// TIA Portal V20 export
DATA_BLOCK "HmiInterface"   // DB93
{ DB_Accessible_From_OPC_UA := 'FALSE' }
AUTHOR : ERsystem_FA2_DH. Kim
// stored: Access Published, DBAccessibleFromOPCUA false, DBAccessibleFromWebserver false, MemoryReserve 100, Namespace Unit1.Em6
   VAR
      em : "LAF_typeEmInterface";
      cm : Struct
         softCam : "Unit1.type_emRelations_em6_SoftCam";
         brakeTest : Struct
            mendrelAnodeFrontAxisZ : "LER_typeBrakeTestEmInterface";
            mendrelAnodeRearAxisZ : "LER_typeBrakeTestEmInterface";
            mendrelCathodeFrontAxisZ : "LER_typeBrakeTestEmInterface";
            mendrelCathodeRearAxisZ : "LER_typeBrakeTestEmInterface";
            stackTableAxisZ : "LER_typeBrakeTestEmInterface";
            stackTableOutFrontAxisZ : "LER_typeBrakeTestEmInterface";
            stackTableOutRearAxisZ : "LER_typeBrakeTestEmInterface";
         END_STRUCT;
         gearIn : Struct
            finalRollerAxisX : "LER_typeGearInInterface";
            stackTableOutAxisZ : "LER_typeGearInInterface";
         END_STRUCT;
      END_STRUCT;
      motion : Struct
         jobs { S7_SetPoint := 'True'} : "LAF_typeJobsInterface";
         sequence { S7_SetPoint := 'True'} : "LAF_typeSequenceInterface";
      END_STRUCT;
      stackTable : Struct
         jobs { S7_SetPoint := 'True'} : "LAF_typeJobsInterface";
         sequence { S7_SetPoint := 'True'} : "LAF_typeSequenceInterface";
      END_STRUCT;
      gaugeRnR : Struct
         jobs { S7_SetPoint := 'True'} : "LAF_typeJobsInterface";
         sequence { S7_SetPoint := 'True'} : "LAF_typeSequenceInterface";
      END_STRUCT;
      utility : Struct
         jobs { S7_SetPoint := 'True'} : "LAF_typeJobsInterface";
         sequence { S7_SetPoint := 'True'} : "LAF_typeSequenceInterface";
      END_STRUCT;
      recipe : Struct
         anodeThickness : LReal := 0.0;
         cathodeThickness : LReal := 0.0;
         sepaThickenss : LReal := 0.0;
         jellyRollThickness : LReal := 0.0;
      END_STRUCT;
      auxiliary : Struct
         parameters : Struct
            finalRollerFrontHomeOffset : LReal := 0.0;
            finalRollerRearHomeOffset : LReal := 0.0;
            stackTableOutFrontHomeOffset : LReal := 0.0;
            stackTableOutRearHomeOffset : LReal := 0.0;
         END_STRUCT;
         commands : Struct
            finalRollerHome : Bool := FALSE;
            stackTableOutHome : Bool := FALSE;
            allMendrelOpen : Bool := FALSE;
            allMendrelClose : Bool := FALSE;
         END_STRUCT;
         monitoring : Struct
            Null : Bool := FALSE;
         END_STRUCT;
      END_STRUCT;
      cmStackTableElectrodeDetect { S7_SetPoint := 'True'} : "LBC_typeDigitalSignalInterface";
   END_VAR
   VAR RETAIN
      cmMasterVirtualAxisX { ExternalVisible := 'False'; ExternalWritable := 'False'} : "LBC_typeAxis64PosInterface";
      cmFinalRollerFrontAxisX { S7_SetPoint := 'True'} : "LBC_typeAxis64PosInterface";
      cmFinalRollerRearAxisX { S7_SetPoint := 'True'} : "LBC_typeAxis64PosInterface";
      cmMendrelAnodeFrontAxisY { S7_SetPoint := 'True'} : "LBC_typeAxis64PosInterface";
      cmMendrelAnodeFrontAxisZ { S7_SetPoint := 'True'} : "LBC_typeAxis64PosInterface";
      cmMendrelAnodeRearAxisY { S7_SetPoint := 'True'} : "LBC_typeAxis64PosInterface";
      cmMendrelAnodeRearAxisZ { S7_SetPoint := 'True'} : "LBC_typeAxis64PosInterface";
      cmMendrelCathodeFrontAxisY : "LBC_typeAxis64PosInterface";
      cmMendrelCathodeFrontAxisZ { S7_SetPoint := 'True'} : "LBC_typeAxis64PosInterface";
      cmMendrelCathodeRearAxisY { S7_SetPoint := 'True'} : "LBC_typeAxis64PosInterface";
      cmMendrelCathodeRearAxisZ { S7_SetPoint := 'True'} : "LBC_typeAxis64PosInterface";
      cmStackTableAxisZ { S7_SetPoint := 'True'} : "LBC_typeAxis64PosInterface";
      cmStackTableOutFrontAxisZ { S7_SetPoint := 'True'} : "LBC_typeAxis64PosInterface";
      cmStackTableOutRearAxisZ { S7_SetPoint := 'True'} : "LBC_typeAxis64PosInterface";
   END_VAR
   VAR
      cmMendrelAnodeFrontClamp { S7_SetPoint := 'True'} : "LBC_typeTwoWayActuatorInterface";
      cmMendrelAnodeRearClamp { S7_SetPoint := 'True'} : "LBC_typeTwoWayActuatorInterface";
      cmMendrelCathodeFrontClamp { S7_SetPoint := 'True'} : "LBC_typeTwoWayActuatorInterface";
      cmMendrelCathodeRearClamp { S7_SetPoint := 'True'} : "LBC_typeTwoWayActuatorInterface";
      cmStackTableVaccum { S7_SetPoint := 'True'} : "LBC_typeTwoWayActuatorInterface";
      cmStackTableGapPadUpDown { S7_SetPoint := 'True'} : "LBC_typeTwoWayActuatorInterface";
      cmStackTableVisionControllerInterface { S7_SetPoint := 'True'} : "LER_typeVisionInterface";
      StackTableVisionConversion : "LER_typeVisionGapResultData";
      StackTableVisionHistory : "LER_typeVisionHistory";
      intCondition : Struct
         Axis_21 { S7_SetPoint := 'True'} : "LER.typeAxisIntlockAll";   // FinalRollerFrontAxisX
         Axis_22 { S7_SetPoint := 'True'} : "LER.typeAxisIntlockAll";   // FinalRollerRearAxisX
         Axis_23 { S7_SetPoint := 'True'} : "LER.typeAxisIntlockAll";   // MandrelFLAxisY
         Axis_24 { S7_SetPoint := 'True'} : "LER.typeAxisIntlockAll";   // MandrelFLAxisZ
         Axis_25 { S7_SetPoint := 'True'} : "LER.typeAxisIntlockAll";   // MandrelFRAxisY
         Axis_26 { S7_SetPoint := 'True'} : "LER.typeAxisIntlockAll";   // MandrelFRAxisZ
         Axis_27 { S7_SetPoint := 'True'} : "LER.typeAxisIntlockAll";   // MandrelRLAxisY
         Axis_28 { S7_SetPoint := 'True'} : "LER.typeAxisIntlockAll";   // MandrelRLAxisZ
         Axis_29 { S7_SetPoint := 'True'} : "LER.typeAxisIntlockAll";   // MandrelRRAxisY
         Axis_30 { S7_SetPoint := 'True'} : "LER.typeAxisIntlockAll";   // MandrelRRAxisZ
         Axis_31 { S7_SetPoint := 'True'} : "LER.typeAxisIntlockAll";   // StackTableAxisZ
         Axis_32 { S7_SetPoint := 'True'} : "LER.typeAxisIntlockAll";   // StackTableOutFrontAxisZ
         Axis_33 { S7_SetPoint := 'True'} : "LER.typeAxisIntlockAll";   // StackTableOutRearAxisZ
         Actuator_33 { S7_SetPoint := 'True'} : "LER.typeAxisActuatorCondition";   // MendrelFLClamp
         Actuator_34 { S7_SetPoint := 'True'} : "LER.typeAxisActuatorCondition";   // MendrelFRClamp
         Actuator_35 { S7_SetPoint := 'True'} : "LER.typeAxisActuatorCondition";   // MendrelRLClamp
         Actuator_36 { S7_SetPoint := 'True'} : "LER.typeAxisActuatorCondition";   // MendrelRRClamp
         Actuator_37 { S7_SetPoint := 'True'} : "LER.typeAxisActuatorCondition";   // StackTableGapPadUpDown
         Actuator_38 { S7_SetPoint := 'True'} : "LER.typeAxisActuatorCondition";   // StackTableGapPadUpDown
      END_STRUCT;
   END_VAR
BEGIN
   em.interlinkMode.link := FALSE;
   em.interlinkMode.unlink := FALSE;
   em.interlinkMode.isLinked := TRUE;
   em.commands.enable := FALSE;
   em.commands.acknowledge := FALSE;
   em.commands.disableAlarms := FALSE;
   em.commands.activateSimulation := FALSE;
   em.commands.home := FALSE;
   em.commands.moveToInitialPosition := FALSE;
   em.commands.directModeControl := 16#0000_0001;
   em.commands.directStateControl := 16#0000_0004;
   em.status.enabled := TRUE;
   em.status.acknowledgeActive := FALSE;
   em.status.alarmsDisabled := FALSE;
   em.status.simulationActive := TRUE;
   em.status.safetyReleased := TRUE;
   em.status.initialized := TRUE;
   em.status.homed := FALSE;
   em.status.safeState := FALSE;
   em.status.stateComplete := FALSE;
   em.alarms.error := FALSE;
   em.alarms.warning := TRUE;
   em.alarms.info := FALSE;
   em.alarms.home := FALSE;
   cm.softCam.finalRollerFrontAxisX.cathode.inPos := FALSE;
   cm.softCam.finalRollerFrontAxisX.cathode.isBefore := FALSE;
   cm.softCam.finalRollerFrontAxisX.cathode.isAfter := TRUE;
   cm.softCam.finalRollerFrontAxisX.anode.inPos := FALSE;
   cm.softCam.finalRollerFrontAxisX.anode.isBefore := TRUE;
   cm.softCam.finalRollerFrontAxisX.anode.isAfter := FALSE;
   cm.softCam.finalRollerFrontAxisX.Pos2.inPos := FALSE;
   cm.softCam.finalRollerFrontAxisX.Pos2.isBefore := FALSE;
   cm.softCam.finalRollerFrontAxisX.Pos2.isAfter := TRUE;
   cm.softCam.finalRollerFrontAxisX.Pos3.inPos := FALSE;
   cm.softCam.finalRollerFrontAxisX.Pos3.isBefore := FALSE;
   cm.softCam.finalRollerFrontAxisX.Pos3.isAfter := TRUE;
   cm.softCam.finalRollerFrontAxisX.Pos4.inPos := FALSE;
   cm.softCam.finalRollerFrontAxisX.Pos4.isBefore := FALSE;
   cm.softCam.finalRollerFrontAxisX.Pos4.isAfter := TRUE;
   cm.softCam.finalRollerFrontAxisX.Pos5.inPos := FALSE;
   cm.softCam.finalRollerFrontAxisX.Pos5.isBefore := FALSE;
   cm.softCam.finalRollerFrontAxisX.Pos5.isAfter := TRUE;
   cm.softCam.finalRollerFrontAxisX.Pos6.inPos := FALSE;
   cm.softCam.finalRollerFrontAxisX.Pos6.isBefore := FALSE;
   cm.softCam.finalRollerFrontAxisX.Pos6.isAfter := TRUE;
   cm.softCam.finalRollerFrontAxisX.Pos7.inPos := FALSE;
   cm.softCam.finalRollerFrontAxisX.Pos7.isBefore := FALSE;
   cm.softCam.finalRollerFrontAxisX.Pos7.isAfter := TRUE;
   cm.softCam.finalRollerFrontAxisX.Pos8.inPos := FALSE;
   cm.softCam.finalRollerFrontAxisX.Pos8.isBefore := FALSE;
   cm.softCam.finalRollerFrontAxisX.Pos8.isAfter := TRUE;
   cm.softCam.finalRollerFrontAxisX.Pos9.inPos := FALSE;
   cm.softCam.finalRollerFrontAxisX.Pos9.isBefore := FALSE;
   cm.softCam.finalRollerFrontAxisX.Pos9.isAfter := TRUE;
   cm.softCam.finalRollerFrontAxisX.Pos10.inPos := FALSE;
   cm.softCam.finalRollerFrontAxisX.Pos10.isBefore := FALSE;
   cm.softCam.finalRollerFrontAxisX.Pos10.isAfter := TRUE;
   cm.softCam.finalRollerFrontAxisX.Pos11.inPos := FALSE;
   cm.softCam.finalRollerFrontAxisX.Pos11.isBefore := FALSE;
   cm.softCam.finalRollerFrontAxisX.Pos11.isAfter := TRUE;
   cm.softCam.finalRollerFrontAxisX.Pos12.inPos := FALSE;
   cm.softCam.finalRollerFrontAxisX.Pos12.isBefore := FALSE;
   cm.softCam.finalRollerFrontAxisX.Pos12.isAfter := TRUE;
   cm.softCam.finalRollerFrontAxisX.Pos13.inPos := FALSE;
   cm.softCam.finalRollerFrontAxisX.Pos13.isBefore := FALSE;
   cm.softCam.finalRollerFrontAxisX.Pos13.isAfter := TRUE;
   cm.softCam.finalRollerFrontAxisX.Pos14.inPos := FALSE;
   cm.softCam.finalRollerFrontAxisX.Pos14.isBefore := FALSE;
   cm.softCam.finalRollerFrontAxisX.Pos14.isAfter := TRUE;
   cm.softCam.finalRollerFrontAxisX.Pos15.inPos := FALSE;
   cm.softCam.finalRollerFrontAxisX.Pos15.isBefore := FALSE;
   cm.softCam.finalRollerFrontAxisX.Pos15.isAfter := TRUE;
   cm.softCam.finalRollerRearAxisX.cathode.inPos := TRUE;
   cm.softCam.finalRollerRearAxisX.cathode.isBefore := FALSE;
   cm.softCam.finalRollerRearAxisX.cathode.isAfter := FALSE;
   cm.softCam.finalRollerRearAxisX.anode.inPos := FALSE;
   cm.softCam.finalRollerRearAxisX.anode.isBefore := TRUE;
   cm.softCam.finalRollerRearAxisX.anode.isAfter := FALSE;
   cm.softCam.finalRollerRearAxisX.Pos2.inPos := TRUE;
   cm.softCam.finalRollerRearAxisX.Pos2.isBefore := FALSE;
   cm.softCam.finalRollerRearAxisX.Pos2.isAfter := FALSE;
   cm.softCam.finalRollerRearAxisX.Pos3.inPos := TRUE;
   cm.softCam.finalRollerRearAxisX.Pos3.isBefore := FALSE;
   cm.softCam.finalRollerRearAxisX.Pos3.isAfter := FALSE;
   cm.softCam.finalRollerRearAxisX.Pos4.inPos := TRUE;
   cm.softCam.finalRollerRearAxisX.Pos4.isBefore := FALSE;
   cm.softCam.finalRollerRearAxisX.Pos4.isAfter := FALSE;
   cm.softCam.finalRollerRearAxisX.Pos5.inPos := TRUE;
   cm.softCam.finalRollerRearAxisX.Pos5.isBefore := FALSE;
   cm.softCam.finalRollerRearAxisX.Pos5.isAfter := FALSE;
   cm.softCam.finalRollerRearAxisX.Pos6.inPos := TRUE;
   cm.softCam.finalRollerRearAxisX.Pos6.isBefore := FALSE;
   cm.softCam.finalRollerRearAxisX.Pos6.isAfter := FALSE;
   cm.softCam.finalRollerRearAxisX.Pos7.inPos := TRUE;
   cm.softCam.finalRollerRearAxisX.Pos7.isBefore := FALSE;
   cm.softCam.finalRollerRearAxisX.Pos7.isAfter := FALSE;
   cm.softCam.finalRollerRearAxisX.Pos8.inPos := TRUE;
   cm.softCam.finalRollerRearAxisX.Pos8.isBefore := FALSE;
   cm.softCam.finalRollerRearAxisX.Pos8.isAfter := FALSE;
   cm.softCam.finalRollerRearAxisX.Pos9.inPos := TRUE;
   cm.softCam.finalRollerRearAxisX.Pos9.isBefore := FALSE;
   cm.softCam.finalRollerRearAxisX.Pos9.isAfter := FALSE;
   cm.softCam.finalRollerRearAxisX.Pos10.inPos := TRUE;
   cm.softCam.finalRollerRearAxisX.Pos10.isBefore := FALSE;
   cm.softCam.finalRollerRearAxisX.Pos10.isAfter := FALSE;
   cm.softCam.finalRollerRearAxisX.Pos11.inPos := TRUE;
   cm.softCam.finalRollerRearAxisX.Pos11.isBefore := FALSE;
   cm.softCam.finalRollerRearAxisX.Pos11.isAfter := FALSE;
   cm.softCam.finalRollerRearAxisX.Pos12.inPos := TRUE;
   cm.softCam.finalRollerRearAxisX.Pos12.isBefore := FALSE;
   cm.softCam.finalRollerRearAxisX.Pos12.isAfter := FALSE;
   cm.softCam.finalRollerRearAxisX.Pos13.inPos := TRUE;
   cm.softCam.finalRollerRearAxisX.Pos13.isBefore := FALSE;
   cm.softCam.finalRollerRearAxisX.Pos13.isAfter := FALSE;
   cm.softCam.finalRollerRearAxisX.Pos14.inPos := TRUE;
   cm.softCam.finalRollerRearAxisX.Pos14.isBefore := FALSE;
   cm.softCam.finalRollerRearAxisX.Pos14.isAfter := FALSE;
   cm.softCam.finalRollerRearAxisX.Pos15.inPos := TRUE;
   cm.softCam.finalRollerRearAxisX.Pos15.isBefore := FALSE;
   cm.softCam.finalRollerRearAxisX.Pos15.isAfter := FALSE;
   cm.softCam.mendrelAnodeFrontAxisY.backward.inPos := FALSE;
   cm.softCam.mendrelAnodeFrontAxisY.backward.isBefore := FALSE;
   cm.softCam.mendrelAnodeFrontAxisY.backward.isAfter := TRUE;
   cm.softCam.mendrelAnodeFrontAxisY.forward.inPos := TRUE;
   cm.softCam.mendrelAnodeFrontAxisY.forward.isBefore := FALSE;
   cm.softCam.mendrelAnodeFrontAxisY.forward.isAfter := FALSE;
   cm.softCam.mendrelAnodeFrontAxisY.Pos2.inPos := FALSE;
   cm.softCam.mendrelAnodeFrontAxisY.Pos2.isBefore := FALSE;
   cm.softCam.mendrelAnodeFrontAxisY.Pos2.isAfter := TRUE;
   cm.softCam.mendrelAnodeFrontAxisY.Pos3.inPos := FALSE;
   cm.softCam.mendrelAnodeFrontAxisY.Pos3.isBefore := FALSE;
   cm.softCam.mendrelAnodeFrontAxisY.Pos3.isAfter := TRUE;
   cm.softCam.mendrelAnodeFrontAxisY.Pos4.inPos := FALSE;
   cm.softCam.mendrelAnodeFrontAxisY.Pos4.isBefore := FALSE;
   cm.softCam.mendrelAnodeFrontAxisY.Pos4.isAfter := TRUE;
   cm.softCam.mendrelAnodeFrontAxisY.Pos5.inPos := FALSE;
   cm.softCam.mendrelAnodeFrontAxisY.Pos5.isBefore := FALSE;
   cm.softCam.mendrelAnodeFrontAxisY.Pos5.isAfter := TRUE;
   cm.softCam.mendrelAnodeFrontAxisY.Pos6.inPos := FALSE;
   cm.softCam.mendrelAnodeFrontAxisY.Pos6.isBefore := FALSE;
   cm.softCam.mendrelAnodeFrontAxisY.Pos6.isAfter := TRUE;
   cm.softCam.mendrelAnodeFrontAxisY.Pos7.inPos := FALSE;
   cm.softCam.mendrelAnodeFrontAxisY.Pos7.isBefore := FALSE;
   cm.softCam.mendrelAnodeFrontAxisY.Pos7.isAfter := TRUE;
   cm.softCam.mendrelAnodeFrontAxisY.Pos8.inPos := FALSE;
   cm.softCam.mendrelAnodeFrontAxisY.Pos8.isBefore := FALSE;
   cm.softCam.mendrelAnodeFrontAxisY.Pos8.isAfter := TRUE;
   cm.softCam.mendrelAnodeFrontAxisY.Pos9.inPos := FALSE;
   cm.softCam.mendrelAnodeFrontAxisY.Pos9.isBefore := FALSE;
   cm.softCam.mendrelAnodeFrontAxisY.Pos9.isAfter := TRUE;
   cm.softCam.mendrelAnodeFrontAxisY.Pos10.inPos := FALSE;
   cm.softCam.mendrelAnodeFrontAxisY.Pos10.isBefore := FALSE;
   cm.softCam.mendrelAnodeFrontAxisY.Pos10.isAfter := TRUE;
   cm.softCam.mendrelAnodeFrontAxisY.Pos11.inPos := FALSE;
   cm.softCam.mendrelAnodeFrontAxisY.Pos11.isBefore := FALSE;
   cm.softCam.mendrelAnodeFrontAxisY.Pos11.isAfter := TRUE;
   cm.softCam.mendrelAnodeFrontAxisY.Pos12.inPos := FALSE;
   cm.softCam.mendrelAnodeFrontAxisY.Pos12.isBefore := FALSE;
   cm.softCam.mendrelAnodeFrontAxisY.Pos12.isAfter := TRUE;
   cm.softCam.mendrelAnodeFrontAxisY.Pos13.inPos := FALSE;
   cm.softCam.mendrelAnodeFrontAxisY.Pos13.isBefore := FALSE;
   cm.softCam.mendrelAnodeFrontAxisY.Pos13.isAfter := TRUE;
   cm.softCam.mendrelAnodeFrontAxisY.Pos14.inPos := FALSE;
   cm.softCam.mendrelAnodeFrontAxisY.Pos14.isBefore := FALSE;
   cm.softCam.mendrelAnodeFrontAxisY.Pos14.isAfter := TRUE;
   cm.softCam.mendrelAnodeFrontAxisY.Pos15.inPos := FALSE;
   cm.softCam.mendrelAnodeFrontAxisY.Pos15.isBefore := FALSE;
   cm.softCam.mendrelAnodeFrontAxisY.Pos15.isAfter := TRUE;
   cm.softCam.mendrelAnodeFrontAxisZ.up.inPos := FALSE;
   cm.softCam.mendrelAnodeFrontAxisZ.up.isBefore := FALSE;
   cm.softCam.mendrelAnodeFrontAxisZ.up.isAfter := TRUE;
   cm.softCam.mendrelAnodeFrontAxisZ.down.inPos := TRUE;
   cm.softCam.mendrelAnodeFrontAxisZ.down.isBefore := FALSE;
   cm.softCam.mendrelAnodeFrontAxisZ.down.isAfter := FALSE;
   cm.softCam.mendrelAnodeFrontAxisZ.Pos2.inPos := FALSE;
   cm.softCam.mendrelAnodeFrontAxisZ.Pos2.isBefore := FALSE;
   cm.softCam.mendrelAnodeFrontAxisZ.Pos2.isAfter := TRUE;
   cm.softCam.mendrelAnodeFrontAxisZ.Pos3.inPos := FALSE;
   cm.softCam.mendrelAnodeFrontAxisZ.Pos3.isBefore := FALSE;
   cm.softCam.mendrelAnodeFrontAxisZ.Pos3.isAfter := TRUE;
   cm.softCam.mendrelAnodeFrontAxisZ.Pos4.inPos := FALSE;
   cm.softCam.mendrelAnodeFrontAxisZ.Pos4.isBefore := FALSE;
   cm.softCam.mendrelAnodeFrontAxisZ.Pos4.isAfter := TRUE;
   cm.softCam.mendrelAnodeFrontAxisZ.Pos5.inPos := FALSE;
   cm.softCam.mendrelAnodeFrontAxisZ.Pos5.isBefore := FALSE;
   cm.softCam.mendrelAnodeFrontAxisZ.Pos5.isAfter := TRUE;
   cm.softCam.mendrelAnodeFrontAxisZ.Pos6.inPos := FALSE;
   cm.softCam.mendrelAnodeFrontAxisZ.Pos6.isBefore := FALSE;
   cm.softCam.mendrelAnodeFrontAxisZ.Pos6.isAfter := TRUE;
   cm.softCam.mendrelAnodeFrontAxisZ.Pos7.inPos := FALSE;
   cm.softCam.mendrelAnodeFrontAxisZ.Pos7.isBefore := FALSE;
   cm.softCam.mendrelAnodeFrontAxisZ.Pos7.isAfter := TRUE;
   cm.softCam.mendrelAnodeFrontAxisZ.Pos8.inPos := FALSE;
   cm.softCam.mendrelAnodeFrontAxisZ.Pos8.isBefore := FALSE;
   cm.softCam.mendrelAnodeFrontAxisZ.Pos8.isAfter := TRUE;
   cm.softCam.mendrelAnodeFrontAxisZ.Pos9.inPos := FALSE;
   cm.softCam.mendrelAnodeFrontAxisZ.Pos9.isBefore := FALSE;
   cm.softCam.mendrelAnodeFrontAxisZ.Pos9.isAfter := TRUE;
   cm.softCam.mendrelAnodeFrontAxisZ.Pos10.inPos := FALSE;
   cm.softCam.mendrelAnodeFrontAxisZ.Pos10.isBefore := FALSE;
   cm.softCam.mendrelAnodeFrontAxisZ.Pos10.isAfter := TRUE;
   cm.softCam.mendrelAnodeFrontAxisZ.Pos11.inPos := FALSE;
   cm.softCam.mendrelAnodeFrontAxisZ.Pos11.isBefore := FALSE;
   cm.softCam.mendrelAnodeFrontAxisZ.Pos11.isAfter := TRUE;
   cm.softCam.mendrelAnodeFrontAxisZ.Pos12.inPos := FALSE;
   cm.softCam.mendrelAnodeFrontAxisZ.Pos12.isBefore := FALSE;
   cm.softCam.mendrelAnodeFrontAxisZ.Pos12.isAfter := TRUE;
   cm.softCam.mendrelAnodeFrontAxisZ.Pos13.inPos := FALSE;
   cm.softCam.mendrelAnodeFrontAxisZ.Pos13.isBefore := FALSE;
   cm.softCam.mendrelAnodeFrontAxisZ.Pos13.isAfter := TRUE;
   cm.softCam.mendrelAnodeFrontAxisZ.Pos14.inPos := FALSE;
   cm.softCam.mendrelAnodeFrontAxisZ.Pos14.isBefore := FALSE;
   cm.softCam.mendrelAnodeFrontAxisZ.Pos14.isAfter := TRUE;
   cm.softCam.mendrelAnodeFrontAxisZ.Pos15.inPos := FALSE;
   cm.softCam.mendrelAnodeFrontAxisZ.Pos15.isBefore := FALSE;
   cm.softCam.mendrelAnodeFrontAxisZ.Pos15.isAfter := TRUE;
   cm.softCam.mendrelAnodeRearAxisY.backward.inPos := FALSE;
   cm.softCam.mendrelAnodeRearAxisY.backward.isBefore := FALSE;
   cm.softCam.mendrelAnodeRearAxisY.backward.isAfter := TRUE;
   cm.softCam.mendrelAnodeRearAxisY.forward.inPos := TRUE;
   cm.softCam.mendrelAnodeRearAxisY.forward.isBefore := FALSE;
   cm.softCam.mendrelAnodeRearAxisY.forward.isAfter := FALSE;
   cm.softCam.mendrelAnodeRearAxisY.Pos2.inPos := FALSE;
   cm.softCam.mendrelAnodeRearAxisY.Pos2.isBefore := FALSE;
   cm.softCam.mendrelAnodeRearAxisY.Pos2.isAfter := TRUE;
   cm.softCam.mendrelAnodeRearAxisY.Pos3.inPos := FALSE;
   cm.softCam.mendrelAnodeRearAxisY.Pos3.isBefore := FALSE;
   cm.softCam.mendrelAnodeRearAxisY.Pos3.isAfter := TRUE;
   cm.softCam.mendrelAnodeRearAxisY.Pos4.inPos := FALSE;
   cm.softCam.mendrelAnodeRearAxisY.Pos4.isBefore := FALSE;
   cm.softCam.mendrelAnodeRearAxisY.Pos4.isAfter := TRUE;
   cm.softCam.mendrelAnodeRearAxisY.Pos5.inPos := FALSE;
   cm.softCam.mendrelAnodeRearAxisY.Pos5.isBefore := FALSE;
   cm.softCam.mendrelAnodeRearAxisY.Pos5.isAfter := TRUE;
   cm.softCam.mendrelAnodeRearAxisY.Pos6.inPos := FALSE;
   cm.softCam.mendrelAnodeRearAxisY.Pos6.isBefore := FALSE;
   cm.softCam.mendrelAnodeRearAxisY.Pos6.isAfter := TRUE;
   cm.softCam.mendrelAnodeRearAxisY.Pos7.inPos := FALSE;
   cm.softCam.mendrelAnodeRearAxisY.Pos7.isBefore := FALSE;
   cm.softCam.mendrelAnodeRearAxisY.Pos7.isAfter := TRUE;
   cm.softCam.mendrelAnodeRearAxisY.Pos8.inPos := FALSE;
   cm.softCam.mendrelAnodeRearAxisY.Pos8.isBefore := FALSE;
   cm.softCam.mendrelAnodeRearAxisY.Pos8.isAfter := TRUE;
   cm.softCam.mendrelAnodeRearAxisY.Pos9.inPos := FALSE;
   cm.softCam.mendrelAnodeRearAxisY.Pos9.isBefore := FALSE;
   cm.softCam.mendrelAnodeRearAxisY.Pos9.isAfter := TRUE;
   cm.softCam.mendrelAnodeRearAxisY.Pos10.inPos := FALSE;
   cm.softCam.mendrelAnodeRearAxisY.Pos10.isBefore := FALSE;
   cm.softCam.mendrelAnodeRearAxisY.Pos10.isAfter := TRUE;
   cm.softCam.mendrelAnodeRearAxisY.Pos11.inPos := FALSE;
   cm.softCam.mendrelAnodeRearAxisY.Pos11.isBefore := FALSE;
   cm.softCam.mendrelAnodeRearAxisY.Pos11.isAfter := TRUE;
   cm.softCam.mendrelAnodeRearAxisY.Pos12.inPos := FALSE;
   cm.softCam.mendrelAnodeRearAxisY.Pos12.isBefore := FALSE;
   cm.softCam.mendrelAnodeRearAxisY.Pos12.isAfter := TRUE;
   cm.softCam.mendrelAnodeRearAxisY.Pos13.inPos := FALSE;
   cm.softCam.mendrelAnodeRearAxisY.Pos13.isBefore := FALSE;
   cm.softCam.mendrelAnodeRearAxisY.Pos13.isAfter := TRUE;
   cm.softCam.mendrelAnodeRearAxisY.Pos14.inPos := FALSE;
   cm.softCam.mendrelAnodeRearAxisY.Pos14.isBefore := FALSE;
   cm.softCam.mendrelAnodeRearAxisY.Pos14.isAfter := TRUE;
   cm.softCam.mendrelAnodeRearAxisY.Pos15.inPos := FALSE;
   cm.softCam.mendrelAnodeRearAxisY.Pos15.isBefore := FALSE;
   cm.softCam.mendrelAnodeRearAxisY.Pos15.isAfter := TRUE;
   cm.softCam.mendrelAnodeRearAxisZ.up.inPos := FALSE;
   cm.softCam.mendrelAnodeRearAxisZ.up.isBefore := FALSE;
   cm.softCam.mendrelAnodeRearAxisZ.up.isAfter := TRUE;
   cm.softCam.mendrelAnodeRearAxisZ.down.inPos := TRUE;
   cm.softCam.mendrelAnodeRearAxisZ.down.isBefore := FALSE;
   cm.softCam.mendrelAnodeRearAxisZ.down.isAfter := FALSE;
   cm.softCam.mendrelAnodeRearAxisZ.Pos2.inPos := FALSE;
   cm.softCam.mendrelAnodeRearAxisZ.Pos2.isBefore := FALSE;
   cm.softCam.mendrelAnodeRearAxisZ.Pos2.isAfter := TRUE;
   cm.softCam.mendrelAnodeRearAxisZ.Pos3.inPos := FALSE;
   cm.softCam.mendrelAnodeRearAxisZ.Pos3.isBefore := FALSE;
   cm.softCam.mendrelAnodeRearAxisZ.Pos3.isAfter := TRUE;
   cm.softCam.mendrelAnodeRearAxisZ.Pos4.inPos := FALSE;
   cm.softCam.mendrelAnodeRearAxisZ.Pos4.isBefore := FALSE;
   cm.softCam.mendrelAnodeRearAxisZ.Pos4.isAfter := TRUE;
   cm.softCam.mendrelAnodeRearAxisZ.Pos5.inPos := FALSE;
   cm.softCam.mendrelAnodeRearAxisZ.Pos5.isBefore := FALSE;
   cm.softCam.mendrelAnodeRearAxisZ.Pos5.isAfter := TRUE;
   cm.softCam.mendrelAnodeRearAxisZ.Pos6.inPos := FALSE;
   cm.softCam.mendrelAnodeRearAxisZ.Pos6.isBefore := FALSE;
   cm.softCam.mendrelAnodeRearAxisZ.Pos6.isAfter := TRUE;
   cm.softCam.mendrelAnodeRearAxisZ.Pos7.inPos := FALSE;
   cm.softCam.mendrelAnodeRearAxisZ.Pos7.isBefore := FALSE;
   cm.softCam.mendrelAnodeRearAxisZ.Pos7.isAfter := TRUE;
   cm.softCam.mendrelAnodeRearAxisZ.Pos8.inPos := FALSE;
   cm.softCam.mendrelAnodeRearAxisZ.Pos8.isBefore := FALSE;
   cm.softCam.mendrelAnodeRearAxisZ.Pos8.isAfter := TRUE;
   cm.softCam.mendrelAnodeRearAxisZ.Pos9.inPos := FALSE;
   cm.softCam.mendrelAnodeRearAxisZ.Pos9.isBefore := FALSE;
   cm.softCam.mendrelAnodeRearAxisZ.Pos9.isAfter := TRUE;
   cm.softCam.mendrelAnodeRearAxisZ.Pos10.inPos := FALSE;
   cm.softCam.mendrelAnodeRearAxisZ.Pos10.isBefore := FALSE;
   cm.softCam.mendrelAnodeRearAxisZ.Pos10.isAfter := TRUE;
   cm.softCam.mendrelAnodeRearAxisZ.Pos11.inPos := FALSE;
   cm.softCam.mendrelAnodeRearAxisZ.Pos11.isBefore := FALSE;
   cm.softCam.mendrelAnodeRearAxisZ.Pos11.isAfter := TRUE;
   cm.softCam.mendrelAnodeRearAxisZ.Pos12.inPos := FALSE;
   cm.softCam.mendrelAnodeRearAxisZ.Pos12.isBefore := FALSE;
   cm.softCam.mendrelAnodeRearAxisZ.Pos12.isAfter := TRUE;
   cm.softCam.mendrelAnodeRearAxisZ.Pos13.inPos := FALSE;
   cm.softCam.mendrelAnodeRearAxisZ.Pos13.isBefore := FALSE;
   cm.softCam.mendrelAnodeRearAxisZ.Pos13.isAfter := TRUE;
   cm.softCam.mendrelAnodeRearAxisZ.Pos14.inPos := FALSE;
   cm.softCam.mendrelAnodeRearAxisZ.Pos14.isBefore := FALSE;
   cm.softCam.mendrelAnodeRearAxisZ.Pos14.isAfter := TRUE;
   cm.softCam.mendrelAnodeRearAxisZ.Pos15.inPos := FALSE;
   cm.softCam.mendrelAnodeRearAxisZ.Pos15.isBefore := FALSE;
   cm.softCam.mendrelAnodeRearAxisZ.Pos15.isAfter := TRUE;
   cm.softCam.mendrelCathodeFrontAxisY.backward.inPos := FALSE;
   cm.softCam.mendrelCathodeFrontAxisY.backward.isBefore := FALSE;
   cm.softCam.mendrelCathodeFrontAxisY.backward.isAfter := TRUE;
   cm.softCam.mendrelCathodeFrontAxisY.forward.inPos := TRUE;
   cm.softCam.mendrelCathodeFrontAxisY.forward.isBefore := FALSE;
   cm.softCam.mendrelCathodeFrontAxisY.forward.isAfter := FALSE;
   cm.softCam.mendrelCathodeFrontAxisY.Pos2.inPos := FALSE;
   cm.softCam.mendrelCathodeFrontAxisY.Pos2.isBefore := FALSE;
   cm.softCam.mendrelCathodeFrontAxisY.Pos2.isAfter := TRUE;
   cm.softCam.mendrelCathodeFrontAxisY.Pos3.inPos := FALSE;
   cm.softCam.mendrelCathodeFrontAxisY.Pos3.isBefore := FALSE;
   cm.softCam.mendrelCathodeFrontAxisY.Pos3.isAfter := TRUE;
   cm.softCam.mendrelCathodeFrontAxisY.Pos4.inPos := FALSE;
   cm.softCam.mendrelCathodeFrontAxisY.Pos4.isBefore := FALSE;
   cm.softCam.mendrelCathodeFrontAxisY.Pos4.isAfter := TRUE;
   cm.softCam.mendrelCathodeFrontAxisY.Pos5.inPos := FALSE;
   cm.softCam.mendrelCathodeFrontAxisY.Pos5.isBefore := FALSE;
   cm.softCam.mendrelCathodeFrontAxisY.Pos5.isAfter := TRUE;
   cm.softCam.mendrelCathodeFrontAxisY.Pos6.inPos := FALSE;
   cm.softCam.mendrelCathodeFrontAxisY.Pos6.isBefore := FALSE;
   cm.softCam.mendrelCathodeFrontAxisY.Pos6.isAfter := TRUE;
   cm.softCam.mendrelCathodeFrontAxisY.Pos7.inPos := FALSE;
   cm.softCam.mendrelCathodeFrontAxisY.Pos7.isBefore := FALSE;
   cm.softCam.mendrelCathodeFrontAxisY.Pos7.isAfter := TRUE;
   cm.softCam.mendrelCathodeFrontAxisY.Pos8.inPos := FALSE;
   cm.softCam.mendrelCathodeFrontAxisY.Pos8.isBefore := FALSE;
   cm.softCam.mendrelCathodeFrontAxisY.Pos8.isAfter := TRUE;
   cm.softCam.mendrelCathodeFrontAxisY.Pos9.inPos := FALSE;
   cm.softCam.mendrelCathodeFrontAxisY.Pos9.isBefore := FALSE;
   cm.softCam.mendrelCathodeFrontAxisY.Pos9.isAfter := TRUE;
   cm.softCam.mendrelCathodeFrontAxisY.Pos10.inPos := FALSE;
   cm.softCam.mendrelCathodeFrontAxisY.Pos10.isBefore := FALSE;
   cm.softCam.mendrelCathodeFrontAxisY.Pos10.isAfter := TRUE;
   cm.softCam.mendrelCathodeFrontAxisY.Pos11.inPos := FALSE;
   cm.softCam.mendrelCathodeFrontAxisY.Pos11.isBefore := FALSE;
   cm.softCam.mendrelCathodeFrontAxisY.Pos11.isAfter := TRUE;
   cm.softCam.mendrelCathodeFrontAxisY.Pos12.inPos := FALSE;
   cm.softCam.mendrelCathodeFrontAxisY.Pos12.isBefore := FALSE;
   cm.softCam.mendrelCathodeFrontAxisY.Pos12.isAfter := TRUE;
   cm.softCam.mendrelCathodeFrontAxisY.Pos13.inPos := FALSE;
   cm.softCam.mendrelCathodeFrontAxisY.Pos13.isBefore := FALSE;
   cm.softCam.mendrelCathodeFrontAxisY.Pos13.isAfter := TRUE;
   cm.softCam.mendrelCathodeFrontAxisY.Pos14.inPos := FALSE;
   cm.softCam.mendrelCathodeFrontAxisY.Pos14.isBefore := FALSE;
   cm.softCam.mendrelCathodeFrontAxisY.Pos14.isAfter := TRUE;
   cm.softCam.mendrelCathodeFrontAxisY.Pos15.inPos := FALSE;
   cm.softCam.mendrelCathodeFrontAxisY.Pos15.isBefore := FALSE;
   cm.softCam.mendrelCathodeFrontAxisY.Pos15.isAfter := TRUE;
   cm.softCam.mendrelCathodeFrontAxisZ.up.inPos := FALSE;
   cm.softCam.mendrelCathodeFrontAxisZ.up.isBefore := FALSE;
   cm.softCam.mendrelCathodeFrontAxisZ.up.isAfter := TRUE;
   cm.softCam.mendrelCathodeFrontAxisZ.down.inPos := TRUE;
   cm.softCam.mendrelCathodeFrontAxisZ.down.isBefore := FALSE;
   cm.softCam.mendrelCathodeFrontAxisZ.down.isAfter := FALSE;
   cm.softCam.mendrelCathodeFrontAxisZ.Pos2.inPos := FALSE;
   cm.softCam.mendrelCathodeFrontAxisZ.Pos2.isBefore := FALSE;
   cm.softCam.mendrelCathodeFrontAxisZ.Pos2.isAfter := TRUE;
   cm.softCam.mendrelCathodeFrontAxisZ.Pos3.inPos := FALSE;
   cm.softCam.mendrelCathodeFrontAxisZ.Pos3.isBefore := FALSE;
   cm.softCam.mendrelCathodeFrontAxisZ.Pos3.isAfter := TRUE;
   cm.softCam.mendrelCathodeFrontAxisZ.Pos4.inPos := FALSE;
   cm.softCam.mendrelCathodeFrontAxisZ.Pos4.isBefore := FALSE;
   cm.softCam.mendrelCathodeFrontAxisZ.Pos4.isAfter := TRUE;
   cm.softCam.mendrelCathodeFrontAxisZ.Pos5.inPos := FALSE;
   cm.softCam.mendrelCathodeFrontAxisZ.Pos5.isBefore := FALSE;
   cm.softCam.mendrelCathodeFrontAxisZ.Pos5.isAfter := TRUE;
   cm.softCam.mendrelCathodeFrontAxisZ.Pos6.inPos := FALSE;
   cm.softCam.mendrelCathodeFrontAxisZ.Pos6.isBefore := FALSE;
   cm.softCam.mendrelCathodeFrontAxisZ.Pos6.isAfter := TRUE;
   cm.softCam.mendrelCathodeFrontAxisZ.Pos7.inPos := FALSE;
   cm.softCam.mendrelCathodeFrontAxisZ.Pos7.isBefore := FALSE;
   cm.softCam.mendrelCathodeFrontAxisZ.Pos7.isAfter := TRUE;
   cm.softCam.mendrelCathodeFrontAxisZ.Pos8.inPos := FALSE;
   cm.softCam.mendrelCathodeFrontAxisZ.Pos8.isBefore := FALSE;
   cm.softCam.mendrelCathodeFrontAxisZ.Pos8.isAfter := TRUE;
   cm.softCam.mendrelCathodeFrontAxisZ.Pos9.inPos := FALSE;
   cm.softCam.mendrelCathodeFrontAxisZ.Pos9.isBefore := FALSE;
   cm.softCam.mendrelCathodeFrontAxisZ.Pos9.isAfter := TRUE;
   cm.softCam.mendrelCathodeFrontAxisZ.Pos10.inPos := FALSE;
   cm.softCam.mendrelCathodeFrontAxisZ.Pos10.isBefore := FALSE;
   cm.softCam.mendrelCathodeFrontAxisZ.Pos10.isAfter := TRUE;
   cm.softCam.mendrelCathodeFrontAxisZ.Pos11.inPos := FALSE;
   cm.softCam.mendrelCathodeFrontAxisZ.Pos11.isBefore := FALSE;
   cm.softCam.mendrelCathodeFrontAxisZ.Pos11.isAfter := TRUE;
   cm.softCam.mendrelCathodeFrontAxisZ.Pos12.inPos := FALSE;
   cm.softCam.mendrelCathodeFrontAxisZ.Pos12.isBefore := FALSE;
   cm.softCam.mendrelCathodeFrontAxisZ.Pos12.isAfter := TRUE;
   cm.softCam.mendrelCathodeFrontAxisZ.Pos13.inPos := FALSE;
   cm.softCam.mendrelCathodeFrontAxisZ.Pos13.isBefore := FALSE;
   cm.softCam.mendrelCathodeFrontAxisZ.Pos13.isAfter := TRUE;
   cm.softCam.mendrelCathodeFrontAxisZ.Pos14.inPos := FALSE;
   cm.softCam.mendrelCathodeFrontAxisZ.Pos14.isBefore := FALSE;
   cm.softCam.mendrelCathodeFrontAxisZ.Pos14.isAfter := TRUE;
   cm.softCam.mendrelCathodeFrontAxisZ.Pos15.inPos := FALSE;
   cm.softCam.mendrelCathodeFrontAxisZ.Pos15.isBefore := FALSE;
   cm.softCam.mendrelCathodeFrontAxisZ.Pos15.isAfter := TRUE;
   cm.softCam.mendrelCathodeRearAxisY.backward.inPos := TRUE;
   cm.softCam.mendrelCathodeRearAxisY.backward.isBefore := FALSE;
   cm.softCam.mendrelCathodeRearAxisY.backward.isAfter := FALSE;
   cm.softCam.mendrelCathodeRearAxisY.forward.inPos := FALSE;
   cm.softCam.mendrelCathodeRearAxisY.forward.isBefore := TRUE;
   cm.softCam.mendrelCathodeRearAxisY.forward.isAfter := FALSE;
   cm.softCam.mendrelCathodeRearAxisY.Pos2.inPos := TRUE;
   cm.softCam.mendrelCathodeRearAxisY.Pos2.isBefore := FALSE;
   cm.softCam.mendrelCathodeRearAxisY.Pos2.isAfter := FALSE;
   cm.softCam.mendrelCathodeRearAxisY.Pos3.inPos := TRUE;
   cm.softCam.mendrelCathodeRearAxisY.Pos3.isBefore := FALSE;
   cm.softCam.mendrelCathodeRearAxisY.Pos3.isAfter := FALSE;
   cm.softCam.mendrelCathodeRearAxisY.Pos4.inPos := TRUE;
   cm.softCam.mendrelCathodeRearAxisY.Pos4.isBefore := FALSE;
   cm.softCam.mendrelCathodeRearAxisY.Pos4.isAfter := FALSE;
   cm.softCam.mendrelCathodeRearAxisY.Pos5.inPos := TRUE;
   cm.softCam.mendrelCathodeRearAxisY.Pos5.isBefore := FALSE;
   cm.softCam.mendrelCathodeRearAxisY.Pos5.isAfter := FALSE;
   cm.softCam.mendrelCathodeRearAxisY.Pos6.inPos := TRUE;
   cm.softCam.mendrelCathodeRearAxisY.Pos6.isBefore := FALSE;
   cm.softCam.mendrelCathodeRearAxisY.Pos6.isAfter := FALSE;
   cm.softCam.mendrelCathodeRearAxisY.Pos7.inPos := TRUE;
   cm.softCam.mendrelCathodeRearAxisY.Pos7.isBefore := FALSE;
   cm.softCam.mendrelCathodeRearAxisY.Pos7.isAfter := FALSE;
   cm.softCam.mendrelCathodeRearAxisY.Pos8.inPos := TRUE;
   cm.softCam.mendrelCathodeRearAxisY.Pos8.isBefore := FALSE;
   cm.softCam.mendrelCathodeRearAxisY.Pos8.isAfter := FALSE;
   cm.softCam.mendrelCathodeRearAxisY.Pos9.inPos := TRUE;
   cm.softCam.mendrelCathodeRearAxisY.Pos9.isBefore := FALSE;
   cm.softCam.mendrelCathodeRearAxisY.Pos9.isAfter := FALSE;
   cm.softCam.mendrelCathodeRearAxisY.Pos10.inPos := TRUE;
   cm.softCam.mendrelCathodeRearAxisY.Pos10.isBefore := FALSE;
   cm.softCam.mendrelCathodeRearAxisY.Pos10.isAfter := FALSE;
   cm.softCam.mendrelCathodeRearAxisY.Pos11.inPos := TRUE;
   cm.softCam.mendrelCathodeRearAxisY.Pos11.isBefore := FALSE;
   cm.softCam.mendrelCathodeRearAxisY.Pos11.isAfter := FALSE;
   cm.softCam.mendrelCathodeRearAxisY.Pos12.inPos := TRUE;
   cm.softCam.mendrelCathodeRearAxisY.Pos12.isBefore := FALSE;
   cm.softCam.mendrelCathodeRearAxisY.Pos12.isAfter := FALSE;
   cm.softCam.mendrelCathodeRearAxisY.Pos13.inPos := TRUE;
   cm.softCam.mendrelCathodeRearAxisY.Pos13.isBefore := FALSE;
   cm.softCam.mendrelCathodeRearAxisY.Pos13.isAfter := FALSE;
   cm.softCam.mendrelCathodeRearAxisY.Pos14.inPos := TRUE;
   cm.softCam.mendrelCathodeRearAxisY.Pos14.isBefore := FALSE;
   cm.softCam.mendrelCathodeRearAxisY.Pos14.isAfter := FALSE;
   cm.softCam.mendrelCathodeRearAxisY.Pos15.inPos := TRUE;
   cm.softCam.mendrelCathodeRearAxisY.Pos15.isBefore := FALSE;
   cm.softCam.mendrelCathodeRearAxisY.Pos15.isAfter := FALSE;
   cm.softCam.mendrelCathodeRearAxisZ.up.inPos := TRUE;
   cm.softCam.mendrelCathodeRearAxisZ.up.isBefore := FALSE;
   cm.softCam.mendrelCathodeRearAxisZ.up.isAfter := FALSE;
   cm.softCam.mendrelCathodeRearAxisZ.down.inPos := FALSE;
   cm.softCam.mendrelCathodeRearAxisZ.down.isBefore := TRUE;
   cm.softCam.mendrelCathodeRearAxisZ.down.isAfter := FALSE;
   cm.softCam.mendrelCathodeRearAxisZ.Pos2.inPos := TRUE;
   cm.softCam.mendrelCathodeRearAxisZ.Pos2.isBefore := FALSE;
   cm.softCam.mendrelCathodeRearAxisZ.Pos2.isAfter := FALSE;
   cm.softCam.mendrelCathodeRearAxisZ.Pos3.inPos := TRUE;
   cm.softCam.mendrelCathodeRearAxisZ.Pos3.isBefore := FALSE;
   cm.softCam.mendrelCathodeRearAxisZ.Pos3.isAfter := FALSE;
   cm.softCam.mendrelCathodeRearAxisZ.Pos4.inPos := TRUE;
   cm.softCam.mendrelCathodeRearAxisZ.Pos4.isBefore := FALSE;
   cm.softCam.mendrelCathodeRearAxisZ.Pos4.isAfter := FALSE;
   cm.softCam.mendrelCathodeRearAxisZ.Pos5.inPos := TRUE;
   cm.softCam.mendrelCathodeRearAxisZ.Pos5.isBefore := FALSE;
   cm.softCam.mendrelCathodeRearAxisZ.Pos5.isAfter := FALSE;
   cm.softCam.mendrelCathodeRearAxisZ.Pos6.inPos := TRUE;
   cm.softCam.mendrelCathodeRearAxisZ.Pos6.isBefore := FALSE;
   cm.softCam.mendrelCathodeRearAxisZ.Pos6.isAfter := FALSE;
   cm.softCam.mendrelCathodeRearAxisZ.Pos7.inPos := TRUE;
   cm.softCam.mendrelCathodeRearAxisZ.Pos7.isBefore := FALSE;
   cm.softCam.mendrelCathodeRearAxisZ.Pos7.isAfter := FALSE;
   cm.softCam.mendrelCathodeRearAxisZ.Pos8.inPos := TRUE;
   cm.softCam.mendrelCathodeRearAxisZ.Pos8.isBefore := FALSE;
   cm.softCam.mendrelCathodeRearAxisZ.Pos8.isAfter := FALSE;
   cm.softCam.mendrelCathodeRearAxisZ.Pos9.inPos := TRUE;
   cm.softCam.mendrelCathodeRearAxisZ.Pos9.isBefore := FALSE;
   cm.softCam.mendrelCathodeRearAxisZ.Pos9.isAfter := FALSE;
   cm.softCam.mendrelCathodeRearAxisZ.Pos10.inPos := TRUE;
   cm.softCam.mendrelCathodeRearAxisZ.Pos10.isBefore := FALSE;
   cm.softCam.mendrelCathodeRearAxisZ.Pos10.isAfter := FALSE;
   cm.softCam.mendrelCathodeRearAxisZ.Pos11.inPos := TRUE;
   cm.softCam.mendrelCathodeRearAxisZ.Pos11.isBefore := FALSE;
   cm.softCam.mendrelCathodeRearAxisZ.Pos11.isAfter := FALSE;
   cm.softCam.mendrelCathodeRearAxisZ.Pos12.inPos := TRUE;
   cm.softCam.mendrelCathodeRearAxisZ.Pos12.isBefore := FALSE;
   cm.softCam.mendrelCathodeRearAxisZ.Pos12.isAfter := FALSE;
   cm.softCam.mendrelCathodeRearAxisZ.Pos13.inPos := TRUE;
   cm.softCam.mendrelCathodeRearAxisZ.Pos13.isBefore := FALSE;
   cm.softCam.mendrelCathodeRearAxisZ.Pos13.isAfter := FALSE;
   cm.softCam.mendrelCathodeRearAxisZ.Pos14.inPos := TRUE;
   cm.softCam.mendrelCathodeRearAxisZ.Pos14.isBefore := FALSE;
   cm.softCam.mendrelCathodeRearAxisZ.Pos14.isAfter := FALSE;
   cm.softCam.mendrelCathodeRearAxisZ.Pos15.inPos := TRUE;
   cm.softCam.mendrelCathodeRearAxisZ.Pos15.isBefore := FALSE;
   cm.softCam.mendrelCathodeRearAxisZ.Pos15.isAfter := FALSE;
   cm.softCam.stackTableAxisZ.wait.inPos := FALSE;
   cm.softCam.stackTableAxisZ.wait.isBefore := TRUE;
   cm.softCam.stackTableAxisZ.wait.isAfter := FALSE;
   cm.softCam.stackTableAxisZ.currentJRThickness.inPos := FALSE;
   cm.softCam.stackTableAxisZ.currentJRThickness.isBefore := TRUE;
   cm.softCam.stackTableAxisZ.currentJRThickness.isAfter := FALSE;
   cm.softCam.stackTableAxisZ.fullJRThickness.inPos := TRUE;
   cm.softCam.stackTableAxisZ.fullJRThickness.isBefore := FALSE;
   cm.softCam.stackTableAxisZ.fullJRThickness.isAfter := FALSE;
   cm.softCam.stackTableAxisZ.Pos3.inPos := TRUE;
   cm.softCam.stackTableAxisZ.Pos3.isBefore := FALSE;
   cm.softCam.stackTableAxisZ.Pos3.isAfter := FALSE;
   cm.softCam.stackTableAxisZ.Pos4.inPos := TRUE;
   cm.softCam.stackTableAxisZ.Pos4.isBefore := FALSE;
   cm.softCam.stackTableAxisZ.Pos4.isAfter := FALSE;
   cm.softCam.stackTableAxisZ.Pos5.inPos := TRUE;
   cm.softCam.stackTableAxisZ.Pos5.isBefore := FALSE;
   cm.softCam.stackTableAxisZ.Pos5.isAfter := FALSE;
   cm.softCam.stackTableAxisZ.Pos6.inPos := TRUE;
   cm.softCam.stackTableAxisZ.Pos6.isBefore := FALSE;
   cm.softCam.stackTableAxisZ.Pos6.isAfter := FALSE;
   cm.softCam.stackTableAxisZ.Pos7.inPos := TRUE;
   cm.softCam.stackTableAxisZ.Pos7.isBefore := FALSE;
   cm.softCam.stackTableAxisZ.Pos7.isAfter := FALSE;
   cm.softCam.stackTableAxisZ.Pos8.inPos := TRUE;
   cm.softCam.stackTableAxisZ.Pos8.isBefore := FALSE;
   cm.softCam.stackTableAxisZ.Pos8.isAfter := FALSE;
   cm.softCam.stackTableAxisZ.Pos9.inPos := TRUE;
   cm.softCam.stackTableAxisZ.Pos9.isBefore := FALSE;
   cm.softCam.stackTableAxisZ.Pos9.isAfter := FALSE;
   cm.softCam.stackTableAxisZ.Pos10.inPos := TRUE;
   cm.softCam.stackTableAxisZ.Pos10.isBefore := FALSE;
   cm.softCam.stackTableAxisZ.Pos10.isAfter := FALSE;
   cm.softCam.stackTableAxisZ.Pos11.inPos := TRUE;
   cm.softCam.stackTableAxisZ.Pos11.isBefore := FALSE;
   cm.softCam.stackTableAxisZ.Pos11.isAfter := FALSE;
   cm.softCam.stackTableAxisZ.Pos12.inPos := TRUE;
   cm.softCam.stackTableAxisZ.Pos12.isBefore := FALSE;
   cm.softCam.stackTableAxisZ.Pos12.isAfter := FALSE;
   cm.softCam.stackTableAxisZ.Pos13.inPos := TRUE;
   cm.softCam.stackTableAxisZ.Pos13.isBefore := FALSE;
   cm.softCam.stackTableAxisZ.Pos13.isAfter := FALSE;
   cm.softCam.stackTableAxisZ.Pos14.inPos := TRUE;
   cm.softCam.stackTableAxisZ.Pos14.isBefore := FALSE;
   cm.softCam.stackTableAxisZ.Pos14.isAfter := FALSE;
   cm.softCam.stackTableAxisZ.Pos15.inPos := TRUE;
   cm.softCam.stackTableAxisZ.Pos15.isBefore := FALSE;
   cm.softCam.stackTableAxisZ.Pos15.isAfter := FALSE;
   cm.softCam.stackTableOutFrontAxisZ.down.inPos := TRUE;
   cm.softCam.stackTableOutFrontAxisZ.down.isBefore := FALSE;
   cm.softCam.stackTableOutFrontAxisZ.down.isAfter := FALSE;
   cm.softCam.stackTableOutFrontAxisZ.up.inPos := FALSE;
   cm.softCam.stackTableOutFrontAxisZ.up.isBefore := TRUE;
   cm.softCam.stackTableOutFrontAxisZ.up.isAfter := FALSE;
   cm.softCam.stackTableOutFrontAxisZ.Pos2.inPos := TRUE;
   cm.softCam.stackTableOutFrontAxisZ.Pos2.isBefore := FALSE;
   cm.softCam.stackTableOutFrontAxisZ.Pos2.isAfter := FALSE;
   cm.softCam.stackTableOutFrontAxisZ.Pos3.inPos := TRUE;
   cm.softCam.stackTableOutFrontAxisZ.Pos3.isBefore := FALSE;
   cm.softCam.stackTableOutFrontAxisZ.Pos3.isAfter := FALSE;
   cm.softCam.stackTableOutFrontAxisZ.Pos4.inPos := TRUE;
   cm.softCam.stackTableOutFrontAxisZ.Pos4.isBefore := FALSE;
   cm.softCam.stackTableOutFrontAxisZ.Pos4.isAfter := FALSE;
   cm.softCam.stackTableOutFrontAxisZ.Pos5.inPos := TRUE;
   cm.softCam.stackTableOutFrontAxisZ.Pos5.isBefore := FALSE;
   cm.softCam.stackTableOutFrontAxisZ.Pos5.isAfter := FALSE;
   cm.softCam.stackTableOutFrontAxisZ.Pos6.inPos := TRUE;
   cm.softCam.stackTableOutFrontAxisZ.Pos6.isBefore := FALSE;
   cm.softCam.stackTableOutFrontAxisZ.Pos6.isAfter := FALSE;
   cm.softCam.stackTableOutFrontAxisZ.Pos7.inPos := TRUE;
   cm.softCam.stackTableOutFrontAxisZ.Pos7.isBefore := FALSE;
   cm.softCam.stackTableOutFrontAxisZ.Pos7.isAfter := FALSE;
   cm.softCam.stackTableOutFrontAxisZ.Pos8.inPos := TRUE;
   cm.softCam.stackTableOutFrontAxisZ.Pos8.isBefore := FALSE;
   cm.softCam.stackTableOutFrontAxisZ.Pos8.isAfter := FALSE;
   cm.softCam.stackTableOutFrontAxisZ.Pos9.inPos := TRUE;
   cm.softCam.stackTableOutFrontAxisZ.Pos9.isBefore := FALSE;
   cm.softCam.stackTableOutFrontAxisZ.Pos9.isAfter := FALSE;
   cm.softCam.stackTableOutFrontAxisZ.Pos10.inPos := TRUE;
   cm.softCam.stackTableOutFrontAxisZ.Pos10.isBefore := FALSE;
   cm.softCam.stackTableOutFrontAxisZ.Pos10.isAfter := FALSE;
   cm.softCam.stackTableOutFrontAxisZ.Pos11.inPos := TRUE;
   cm.softCam.stackTableOutFrontAxisZ.Pos11.isBefore := FALSE;
   cm.softCam.stackTableOutFrontAxisZ.Pos11.isAfter := FALSE;
   cm.softCam.stackTableOutFrontAxisZ.Pos12.inPos := TRUE;
   cm.softCam.stackTableOutFrontAxisZ.Pos12.isBefore := FALSE;
   cm.softCam.stackTableOutFrontAxisZ.Pos12.isAfter := FALSE;
   cm.softCam.stackTableOutFrontAxisZ.Pos13.inPos := TRUE;
   cm.softCam.stackTableOutFrontAxisZ.Pos13.isBefore := FALSE;
   cm.softCam.stackTableOutFrontAxisZ.Pos13.isAfter := FALSE;
   cm.softCam.stackTableOutFrontAxisZ.Pos14.inPos := TRUE;
   cm.softCam.stackTableOutFrontAxisZ.Pos14.isBefore := FALSE;
   cm.softCam.stackTableOutFrontAxisZ.Pos14.isAfter := FALSE;
   cm.softCam.stackTableOutFrontAxisZ.Pos15.inPos := TRUE;
   cm.softCam.stackTableOutFrontAxisZ.Pos15.isBefore := FALSE;
   cm.softCam.stackTableOutFrontAxisZ.Pos15.isAfter := FALSE;
   cm.softCam.stackTableOutRearAxisZ.down.inPos := TRUE;
   cm.softCam.stackTableOutRearAxisZ.down.isBefore := FALSE;
   cm.softCam.stackTableOutRearAxisZ.down.isAfter := FALSE;
   cm.softCam.stackTableOutRearAxisZ.up.inPos := FALSE;
   cm.softCam.stackTableOutRearAxisZ.up.isBefore := TRUE;
   cm.softCam.stackTableOutRearAxisZ.up.isAfter := FALSE;
   cm.softCam.stackTableOutRearAxisZ.Pos2.inPos := TRUE;
   cm.softCam.stackTableOutRearAxisZ.Pos2.isBefore := FALSE;
   cm.softCam.stackTableOutRearAxisZ.Pos2.isAfter := FALSE;
   cm.softCam.stackTableOutRearAxisZ.Pos3.inPos := TRUE;
   cm.softCam.stackTableOutRearAxisZ.Pos3.isBefore := FALSE;
   cm.softCam.stackTableOutRearAxisZ.Pos3.isAfter := FALSE;
   cm.softCam.stackTableOutRearAxisZ.Pos4.inPos := TRUE;
   cm.softCam.stackTableOutRearAxisZ.Pos4.isBefore := FALSE;
   cm.softCam.stackTableOutRearAxisZ.Pos4.isAfter := FALSE;
   cm.softCam.stackTableOutRearAxisZ.Pos5.inPos := TRUE;
   cm.softCam.stackTableOutRearAxisZ.Pos5.isBefore := FALSE;
   cm.softCam.stackTableOutRearAxisZ.Pos5.isAfter := FALSE;
   cm.softCam.stackTableOutRearAxisZ.Pos6.inPos := TRUE;
   cm.softCam.stackTableOutRearAxisZ.Pos6.isBefore := FALSE;
   cm.softCam.stackTableOutRearAxisZ.Pos6.isAfter := FALSE;
   cm.softCam.stackTableOutRearAxisZ.Pos7.inPos := TRUE;
   cm.softCam.stackTableOutRearAxisZ.Pos7.isBefore := FALSE;
   cm.softCam.stackTableOutRearAxisZ.Pos7.isAfter := FALSE;
   cm.softCam.stackTableOutRearAxisZ.Pos8.inPos := TRUE;
   cm.softCam.stackTableOutRearAxisZ.Pos8.isBefore := FALSE;
   cm.softCam.stackTableOutRearAxisZ.Pos8.isAfter := FALSE;
   cm.softCam.stackTableOutRearAxisZ.Pos9.inPos := TRUE;
   cm.softCam.stackTableOutRearAxisZ.Pos9.isBefore := FALSE;
   cm.softCam.stackTableOutRearAxisZ.Pos9.isAfter := FALSE;
   cm.softCam.stackTableOutRearAxisZ.Pos10.inPos := TRUE;
   cm.softCam.stackTableOutRearAxisZ.Pos10.isBefore := FALSE;
   cm.softCam.stackTableOutRearAxisZ.Pos10.isAfter := FALSE;
   cm.softCam.stackTableOutRearAxisZ.Pos11.inPos := TRUE;
   cm.softCam.stackTableOutRearAxisZ.Pos11.isBefore := FALSE;
   cm.softCam.stackTableOutRearAxisZ.Pos11.isAfter := FALSE;
   cm.softCam.stackTableOutRearAxisZ.Pos12.inPos := TRUE;
   cm.softCam.stackTableOutRearAxisZ.Pos12.isBefore := FALSE;
   cm.softCam.stackTableOutRearAxisZ.Pos12.isAfter := FALSE;
   cm.softCam.stackTableOutRearAxisZ.Pos13.inPos := TRUE;
   cm.softCam.stackTableOutRearAxisZ.Pos13.isBefore := FALSE;
   cm.softCam.stackTableOutRearAxisZ.Pos13.isAfter := FALSE;
   cm.softCam.stackTableOutRearAxisZ.Pos14.inPos := TRUE;
   cm.softCam.stackTableOutRearAxisZ.Pos14.isBefore := FALSE;
   cm.softCam.stackTableOutRearAxisZ.Pos14.isAfter := FALSE;
   cm.softCam.stackTableOutRearAxisZ.Pos15.inPos := TRUE;
   cm.softCam.stackTableOutRearAxisZ.Pos15.isBefore := FALSE;
   cm.softCam.stackTableOutRearAxisZ.Pos15.isAfter := FALSE;
   cm.brakeTest.mendrelAnodeFrontAxisZ.commands.start := FALSE;
   cm.brakeTest.mendrelAnodeFrontAxisZ.commands.stop := FALSE;
   cm.brakeTest.mendrelAnodeFrontAxisZ.monitoring.error := FALSE;
   cm.brakeTest.mendrelAnodeFrontAxisZ.monitoring.ready := FALSE;
   cm.brakeTest.mendrelAnodeFrontAxisZ.monitoring.busy := FALSE;
   cm.brakeTest.mendrelAnodeFrontAxisZ.monitoring.complete := FALSE;
   cm.brakeTest.mendrelAnodeFrontAxisZ.monitoring.brakeSelected := FALSE;
   cm.brakeTest.mendrelAnodeFrontAxisZ.monitoring.brakeActive := FALSE;
   cm.brakeTest.mendrelAnodeFrontAxisZ.monitoring.brakeResult := FALSE;
   cm.brakeTest.mendrelAnodeFrontAxisZ.monitoring.brakeCompleted := FALSE;
   cm.brakeTest.mendrelAnodeFrontAxisZ.monitoring."step" := 0;
   cm.brakeTest.mendrelAnodeRearAxisZ.commands.start := FALSE;
   cm.brakeTest.mendrelAnodeRearAxisZ.commands.stop := FALSE;
   cm.brakeTest.mendrelAnodeRearAxisZ.monitoring.error := FALSE;
   cm.brakeTest.mendrelAnodeRearAxisZ.monitoring.ready := FALSE;
   cm.brakeTest.mendrelAnodeRearAxisZ.monitoring.busy := FALSE;
   cm.brakeTest.mendrelAnodeRearAxisZ.monitoring.complete := FALSE;
   cm.brakeTest.mendrelAnodeRearAxisZ.monitoring.brakeSelected := FALSE;
   cm.brakeTest.mendrelAnodeRearAxisZ.monitoring.brakeActive := FALSE;
   cm.brakeTest.mendrelAnodeRearAxisZ.monitoring.brakeResult := FALSE;
   cm.brakeTest.mendrelAnodeRearAxisZ.monitoring.brakeCompleted := FALSE;
   cm.brakeTest.mendrelAnodeRearAxisZ.monitoring."step" := 0;
   cm.brakeTest.mendrelCathodeFrontAxisZ.commands.start := FALSE;
   cm.brakeTest.mendrelCathodeFrontAxisZ.commands.stop := FALSE;
   cm.brakeTest.mendrelCathodeFrontAxisZ.monitoring.error := FALSE;
   cm.brakeTest.mendrelCathodeFrontAxisZ.monitoring.ready := FALSE;
   cm.brakeTest.mendrelCathodeFrontAxisZ.monitoring.busy := FALSE;
   cm.brakeTest.mendrelCathodeFrontAxisZ.monitoring.complete := FALSE;
   cm.brakeTest.mendrelCathodeFrontAxisZ.monitoring.brakeSelected := FALSE;
   cm.brakeTest.mendrelCathodeFrontAxisZ.monitoring.brakeActive := FALSE;
   cm.brakeTest.mendrelCathodeFrontAxisZ.monitoring.brakeResult := FALSE;
   cm.brakeTest.mendrelCathodeFrontAxisZ.monitoring.brakeCompleted := FALSE;
   cm.brakeTest.mendrelCathodeFrontAxisZ.monitoring."step" := 0;
   cm.brakeTest.mendrelCathodeRearAxisZ.commands.start := FALSE;
   cm.brakeTest.mendrelCathodeRearAxisZ.commands.stop := FALSE;
   cm.brakeTest.mendrelCathodeRearAxisZ.monitoring.error := FALSE;
   cm.brakeTest.mendrelCathodeRearAxisZ.monitoring.ready := FALSE;
   cm.brakeTest.mendrelCathodeRearAxisZ.monitoring.busy := FALSE;
   cm.brakeTest.mendrelCathodeRearAxisZ.monitoring.complete := FALSE;
   cm.brakeTest.mendrelCathodeRearAxisZ.monitoring.brakeSelected := FALSE;
   cm.brakeTest.mendrelCathodeRearAxisZ.monitoring.brakeActive := FALSE;
   cm.brakeTest.mendrelCathodeRearAxisZ.monitoring.brakeResult := FALSE;
   cm.brakeTest.mendrelCathodeRearAxisZ.monitoring.brakeCompleted := FALSE;
   cm.brakeTest.mendrelCathodeRearAxisZ.monitoring."step" := 0;
   cm.brakeTest.stackTableAxisZ.commands.start := FALSE;
   cm.brakeTest.stackTableAxisZ.commands.stop := FALSE;
   cm.brakeTest.stackTableAxisZ.monitoring.error := FALSE;
   cm.brakeTest.stackTableAxisZ.monitoring.ready := FALSE;
   cm.brakeTest.stackTableAxisZ.monitoring.busy := FALSE;
   cm.brakeTest.stackTableAxisZ.monitoring.complete := FALSE;
   cm.brakeTest.stackTableAxisZ.monitoring.brakeSelected := FALSE;
   cm.brakeTest.stackTableAxisZ.monitoring.brakeActive := FALSE;
   cm.brakeTest.stackTableAxisZ.monitoring.brakeResult := FALSE;
   cm.brakeTest.stackTableAxisZ.monitoring.brakeCompleted := FALSE;
   cm.brakeTest.stackTableAxisZ.monitoring."step" := 0;
   cm.brakeTest.stackTableOutFrontAxisZ.commands.start := FALSE;
   cm.brakeTest.stackTableOutFrontAxisZ.commands.stop := FALSE;
   cm.brakeTest.stackTableOutFrontAxisZ.monitoring.error := FALSE;
   cm.brakeTest.stackTableOutFrontAxisZ.monitoring.ready := FALSE;
   cm.brakeTest.stackTableOutFrontAxisZ.monitoring.busy := FALSE;
   cm.brakeTest.stackTableOutFrontAxisZ.monitoring.complete := FALSE;
   cm.brakeTest.stackTableOutFrontAxisZ.monitoring.brakeSelected := FALSE;
   cm.brakeTest.stackTableOutFrontAxisZ.monitoring.brakeActive := FALSE;
   cm.brakeTest.stackTableOutFrontAxisZ.monitoring.brakeResult := FALSE;
   cm.brakeTest.stackTableOutFrontAxisZ.monitoring.brakeCompleted := FALSE;
   cm.brakeTest.stackTableOutFrontAxisZ.monitoring."step" := 0;
   cm.brakeTest.stackTableOutRearAxisZ.commands.start := FALSE;
   cm.brakeTest.stackTableOutRearAxisZ.commands.stop := FALSE;
   cm.brakeTest.stackTableOutRearAxisZ.monitoring.error := FALSE;
   cm.brakeTest.stackTableOutRearAxisZ.monitoring.ready := FALSE;
   cm.brakeTest.stackTableOutRearAxisZ.monitoring.busy := FALSE;
   cm.brakeTest.stackTableOutRearAxisZ.monitoring.complete := FALSE;
   cm.brakeTest.stackTableOutRearAxisZ.monitoring.brakeSelected := FALSE;
   cm.brakeTest.stackTableOutRearAxisZ.monitoring.brakeActive := FALSE;
   cm.brakeTest.stackTableOutRearAxisZ.monitoring.brakeResult := FALSE;
   cm.brakeTest.stackTableOutRearAxisZ.monitoring.brakeCompleted := FALSE;
   cm.brakeTest.stackTableOutRearAxisZ.monitoring."step" := 0;
   motion.jobs.commands.setJobNumber := 0;
   motion.jobs.commands.reset := FALSE;
   motion.jobs.status.activeJobNumber := 0;
   motion.jobs.status.previousCycleJobNumber := 0;
   motion.jobs.status.manualControlEnabled := FALSE;
   motion.jobs.status.memoryJobTime := 0.0;
   motion.sequence.commands.setAutomaticMode := FALSE;
   motion.sequence.commands.setSingleStepMode := FALSE;
   motion.sequence.commands.off := FALSE;
   motion.sequence.commands.initialize := FALSE;
   motion.sequence.commands.start := FALSE;
   motion.sequence.commands.immediateStop := FALSE;
   motion.sequence.commands.hold := FALSE;
   motion.sequence.commands.nextStep := FALSE;
   motion.sequence.commands.interlockStepChange := FALSE;
   motion.sequence.monitoring.automaticMode := FALSE;
   motion.sequence.monitoring.singleStepMode := FALSE;
   motion.sequence.monitoring.currentStep := 0;
   motion.sequence.monitoring.nextStep := 0;
   motion.sequence.monitoring.previousStep := 0;
   motion.sequence.monitoring.currentStepSTRING := '';
   motion.sequence.monitoring.nextStepSTRING := '';
   motion.sequence.monitoring.previousStepSTRING := '';
   motion.sequence.monitoring.inStepIdle := FALSE;
   motion.sequence.monitoring.inStepStopped := FALSE;
   motion.sequence.monitoring.seqActive := FALSE;
   motion.sequence.monitoring.stepActive := FALSE;
   motion.sequence.monitoring.stepComplete := FALSE;
   motion.sequence.monitoring.executionEnabled := FALSE;
   motion.sequence.monitoring.initRequired := FALSE;
   motion.sequence.monitoring.stepChangeReleased := FALSE;
   motion.sequence.monitoring.justSteppedPulse := FALSE;
   motion.sequence.monitoring.manualControlEnabled := FALSE;
   motion.sequence.monitoring.manualModeChangeEnabled := FALSE;
   motion.sequence.monitoring.memoryStepTimer := 0.0;
   stackTable.jobs.commands.setJobNumber := 0;
   stackTable.jobs.commands.reset := FALSE;
   stackTable.jobs.status.activeJobNumber := 0;
   stackTable.jobs.status.previousCycleJobNumber := 0;
   stackTable.jobs.status.manualControlEnabled := FALSE;
   stackTable.jobs.status.memoryJobTime := 16#0000_4EB8_1052_0721;
   stackTable.sequence.commands.setAutomaticMode := FALSE;
   stackTable.sequence.commands.setSingleStepMode := FALSE;
   stackTable.sequence.commands.off := FALSE;
   stackTable.sequence.commands.initialize := FALSE;
   stackTable.sequence.commands.start := FALSE;
   stackTable.sequence.commands.immediateStop := FALSE;
   stackTable.sequence.commands.hold := FALSE;
   stackTable.sequence.commands.nextStep := FALSE;
   stackTable.sequence.commands.interlockStepChange := FALSE;
   stackTable.sequence.monitoring.automaticMode := TRUE;
   stackTable.sequence.monitoring.singleStepMode := FALSE;
   stackTable.sequence.monitoring.currentStep := 1;
   stackTable.sequence.monitoring.nextStep := 1;
   stackTable.sequence.monitoring.previousStep := 190;
   stackTable.sequence.monitoring.currentStepSTRING := 'N/A';
   stackTable.sequence.monitoring.nextStepSTRING := 'N/A';
   stackTable.sequence.monitoring.previousStepSTRING := 'N/A';
   stackTable.sequence.monitoring.inStepIdle := TRUE;
   stackTable.sequence.monitoring.inStepStopped := FALSE;
   stackTable.sequence.monitoring.seqActive := TRUE;
   stackTable.sequence.monitoring.stepActive := TRUE;
   stackTable.sequence.monitoring.stepComplete := FALSE;
   stackTable.sequence.monitoring.executionEnabled := TRUE;
   stackTable.sequence.monitoring.initRequired := FALSE;
   stackTable.sequence.monitoring.stepChangeReleased := TRUE;
   stackTable.sequence.monitoring.justSteppedPulse := FALSE;
   stackTable.sequence.monitoring.manualControlEnabled := FALSE;
   stackTable.sequence.monitoring.manualModeChangeEnabled := FALSE;
   stackTable.sequence.monitoring.memoryStepTimer := 16#0000_4EB8_1051_50A2;
   gaugeRnR.jobs.commands.setJobNumber := 0;
   gaugeRnR.jobs.commands.reset := FALSE;
   gaugeRnR.jobs.status.activeJobNumber := 0;
   gaugeRnR.jobs.status.previousCycleJobNumber := 0;
   gaugeRnR.jobs.status.manualControlEnabled := FALSE;
   gaugeRnR.jobs.status.memoryJobTime := 0.0;
   gaugeRnR.sequence.commands.setAutomaticMode := FALSE;
   gaugeRnR.sequence.commands.setSingleStepMode := FALSE;
   gaugeRnR.sequence.commands.off := FALSE;
   gaugeRnR.sequence.commands.initialize := FALSE;
   gaugeRnR.sequence.commands.start := FALSE;
   gaugeRnR.sequence.commands.immediateStop := FALSE;
   gaugeRnR.sequence.commands.hold := FALSE;
   gaugeRnR.sequence.commands.nextStep := FALSE;
   gaugeRnR.sequence.commands.interlockStepChange := FALSE;
   gaugeRnR.sequence.monitoring.automaticMode := FALSE;
   gaugeRnR.sequence.monitoring.singleStepMode := FALSE;
   gaugeRnR.sequence.monitoring.currentStep := 0;
   gaugeRnR.sequence.monitoring.nextStep := 0;
   gaugeRnR.sequence.monitoring.previousStep := 0;
   gaugeRnR.sequence.monitoring.currentStepSTRING := 'N/A';
   gaugeRnR.sequence.monitoring.nextStepSTRING := 'N/A';
   gaugeRnR.sequence.monitoring.previousStepSTRING := 'N/A';
   gaugeRnR.sequence.monitoring.inStepIdle := FALSE;
   gaugeRnR.sequence.monitoring.inStepStopped := FALSE;
   gaugeRnR.sequence.monitoring.seqActive := TRUE;
   gaugeRnR.sequence.monitoring.stepActive := TRUE;
   gaugeRnR.sequence.monitoring.stepComplete := FALSE;
   gaugeRnR.sequence.monitoring.executionEnabled := FALSE;
   gaugeRnR.sequence.monitoring.initRequired := FALSE;
   gaugeRnR.sequence.monitoring.stepChangeReleased := FALSE;
   gaugeRnR.sequence.monitoring.justSteppedPulse := FALSE;
   gaugeRnR.sequence.monitoring.manualControlEnabled := FALSE;
   gaugeRnR.sequence.monitoring.manualModeChangeEnabled := FALSE;
   gaugeRnR.sequence.monitoring.memoryStepTimer := 0.0;
   utility.jobs.commands.setJobNumber := 0;
   utility.jobs.commands.reset := FALSE;
   utility.jobs.status.activeJobNumber := 0;
   utility.jobs.status.previousCycleJobNumber := 0;
   utility.jobs.status.manualControlEnabled := FALSE;
   utility.jobs.status.memoryJobTime := 0.0;
   utility.sequence.commands.setAutomaticMode := FALSE;
   utility.sequence.commands.setSingleStepMode := FALSE;
   utility.sequence.commands.off := FALSE;
   utility.sequence.commands.initialize := FALSE;
   utility.sequence.commands.start := FALSE;
   utility.sequence.commands.immediateStop := FALSE;
   utility.sequence.commands.hold := FALSE;
   utility.sequence.commands.nextStep := FALSE;
   utility.sequence.commands.interlockStepChange := FALSE;
   utility.sequence.monitoring.automaticMode := FALSE;
   utility.sequence.monitoring.singleStepMode := FALSE;
   utility.sequence.monitoring.currentStep := 0;
   utility.sequence.monitoring.nextStep := 0;
   utility.sequence.monitoring.previousStep := 0;
   utility.sequence.monitoring.currentStepSTRING := 'N/A';
   utility.sequence.monitoring.nextStepSTRING := 'N/A';
   utility.sequence.monitoring.previousStepSTRING := 'N/A';
   utility.sequence.monitoring.inStepIdle := FALSE;
   utility.sequence.monitoring.inStepStopped := FALSE;
   utility.sequence.monitoring.seqActive := TRUE;
   utility.sequence.monitoring.stepActive := TRUE;
   utility.sequence.monitoring.stepComplete := FALSE;
   utility.sequence.monitoring.executionEnabled := FALSE;
   utility.sequence.monitoring.initRequired := FALSE;
   utility.sequence.monitoring.stepChangeReleased := FALSE;
   utility.sequence.monitoring.justSteppedPulse := FALSE;
   utility.sequence.monitoring.manualControlEnabled := FALSE;
   utility.sequence.monitoring.manualModeChangeEnabled := FALSE;
   utility.sequence.monitoring.memoryStepTimer := 0.0;
   cmStackTableElectrodeDetect.commands.refreshConfiguration := FALSE;
   cmStackTableElectrodeDetect.commands.editConfiguration := FALSE;
   cmStackTableElectrodeDetect.commands.saveConfiguration := FALSE;
   cmStackTableElectrodeDetect.commands.reset := FALSE;
   cmStackTableElectrodeDetect.monitoring.enable := TRUE;
   cmStackTableElectrodeDetect.monitoring.referenceDesignator := WSTRING#'DigitalSignal';
   cmStackTableElectrodeDetect.monitoring.simulation := FALSE;
   cmStackTableElectrodeDetect.monitoring.processValue := FALSE;
   cmStackTableElectrodeDetect.monitoring.error := FALSE;
   cmStackTableElectrodeDetect.monitoring.status := 16#0000;
   cmStackTableElectrodeDetect.configuration.referenceDesignator := WSTRING#'DigitalSignal';
   cmStackTableElectrodeDetect.configuration.onDelay := T#0MS;
   cmStackTableElectrodeDetect.configuration.offDelay := T#0MS;
   cmStackTableElectrodeDetect.configuration.default := FALSE;
   cmStackTableElectrodeDetect.configuration.invertProcessValue := FALSE;
   cmStackTableElectrodeDetect.configuration.disableAlarms := FALSE;
   cmMasterVirtualAxisX.commandConfiguration.generalSettings.stopOnError := TRUE;
   cmMasterVirtualAxisX.commandConfiguration.generalSettings.resetWithRestart := FALSE;
   cmMasterVirtualAxisX.commandConfiguration.generalSettings.abortWaitingSyncCmd := TRUE;
   cmMasterVirtualAxisX.commandConfiguration.power.startMode := 1;
   cmMasterVirtualAxisX.commandConfiguration.power.stopMode := 0;
   cmMasterVirtualAxisX.commandConfiguration.power.syncMotionSimulation := FALSE;
   cmMasterVirtualAxisX.commandConfiguration.power.syncMotionSimulationExtendedMode := -1;
   cmMasterVirtualAxisX.commandConfiguration.jog.velocity := 0.0;
   cmMasterVirtualAxisX.commandConfiguration.jog.acceleration := -1.0;
   cmMasterVirtualAxisX.commandConfiguration.jog.deceleration := -1.0;
   cmMasterVirtualAxisX.commandConfiguration.jog.jerk := -1.0;
   cmMasterVirtualAxisX.commandConfiguration.jog.positionControlled := TRUE;
   cmMasterVirtualAxisX.commandConfiguration.jog.increment := 0.0;
   cmMasterVirtualAxisX.commandConfiguration.jog.mode := 0;
   cmMasterVirtualAxisX.commandConfiguration.moveVelocity.velocity := 0.0;
   cmMasterVirtualAxisX.commandConfiguration.moveVelocity.acceleration := -1.0;
   cmMasterVirtualAxisX.commandConfiguration.moveVelocity.deceleration := -1.0;
   cmMasterVirtualAxisX.commandConfiguration.moveVelocity.jerk := -1.0;
   cmMasterVirtualAxisX.commandConfiguration.moveVelocity.direction := 0;
   cmMasterVirtualAxisX.commandConfiguration.moveVelocity.positionControlled := TRUE;
   cmMasterVirtualAxisX.commandConfiguration.moveVelocity.velocityChangeOnTheFly := FALSE;
   cmMasterVirtualAxisX.commandConfiguration.stop.deceleration := -1.0;
   cmMasterVirtualAxisX.commandConfiguration.stop.jerk := -1.0;
   cmMasterVirtualAxisX.commandConfiguration.stop.abortAcceleration := FALSE;
   cmMasterVirtualAxisX.commandConfiguration.fastStop.deceleration := -1.0;
   cmMasterVirtualAxisX.commandConfiguration.fastStop.jerk := -1.0;
   cmMasterVirtualAxisX.commandConfiguration.fastStop.abortAcceleration := FALSE;
   cmMasterVirtualAxisX.commandConfiguration.fastStop.replaceStopPossible := FALSE;
   cmMasterVirtualAxisX.commandConfiguration.torqueLimiting.limit := -1.0;
   cmMasterVirtualAxisX.commandConfiguration.torqueLimiting.mode := 0;
   cmMasterVirtualAxisX.commandConfiguration.homing.position := 0.0;
   cmMasterVirtualAxisX.commandConfiguration.homing.mode := 0;
   cmMasterVirtualAxisX.commandConfiguration.homing.sensor := 0;
   cmMasterVirtualAxisX.commandConfiguration.homing.extendedMode := -1;
   cmMasterVirtualAxisX.commandConfiguration.homing.extendedModeTorqueLimit := 0.0;
   cmMasterVirtualAxisX.commandConfiguration.homing.extendedModeTargetPosition := 0.0;
   cmMasterVirtualAxisX.commandConfiguration.posRelative.distance := 0.0;
   cmMasterVirtualAxisX.commandConfiguration.posRelative.velocity := -1.0;
   cmMasterVirtualAxisX.commandConfiguration.posRelative.acceleration := -1.0;
   cmMasterVirtualAxisX.commandConfiguration.posRelative.deceleration := -1.0;
   cmMasterVirtualAxisX.commandConfiguration.posRelative.jerk := -1.0;
   cmMasterVirtualAxisX.commandConfiguration.posRelative.direction := 0;
   cmMasterVirtualAxisX.commandConfiguration.posAbsolute.position := 0.0;
   cmMasterVirtualAxisX.commandConfiguration.posAbsolute.velocity := -1.0;
   cmMasterVirtualAxisX.commandConfiguration.posAbsolute.acceleration := -1.0;
   cmMasterVirtualAxisX.commandConfiguration.posAbsolute.deceleration := -1.0;
   cmMasterVirtualAxisX.commandConfiguration.posAbsolute.jerk := -1.0;
   cmMasterVirtualAxisX.commandConfiguration.posAbsolute.direction := 1;
   cmMasterVirtualAxisX.commandConfiguration.posAbsolute.positionChangeOnTheFly := FALSE;
   cmMasterVirtualAxisX.commandConfiguration.posAbsolute.velocityChangeOnTheFly := FALSE;
   cmMasterVirtualAxisX.commandConfiguration.posSuperimposed.distance := 0.0;
   cmMasterVirtualAxisX.commandConfiguration.posSuperimposed.velocityDiff := -1.0;
   cmMasterVirtualAxisX.commandConfiguration.posSuperimposed.acceleration := -1.0;
   cmMasterVirtualAxisX.commandConfiguration.posSuperimposed.deceleration := -1.0;
   cmMasterVirtualAxisX.commandConfiguration.posSuperimposed.jerk := -1.0;
   cmMasterVirtualAxisX.commandConfiguration.posSuperimposed.direction := 0;
   cmMasterVirtualAxisX.commandConfiguration.haltSuperimposed.deceleration := -1.0;
   cmMasterVirtualAxisX.commandConfiguration.haltSuperimposed.jerk := -1.0;
   cmMasterVirtualAxisX.commandConfiguration.haltSuperimposed.abortAcceleration := FALSE;
   cmMasterVirtualAxisX.commandConfiguration.gearInRelative.ratioNumerator := 1;
   cmMasterVirtualAxisX.commandConfiguration.gearInRelative.ratioDenominator := 1;
   cmMasterVirtualAxisX.commandConfiguration.gearInRelative.acceleration := -1.0;
   cmMasterVirtualAxisX.commandConfiguration.gearInRelative.deceleration := -1.0;
   cmMasterVirtualAxisX.commandConfiguration.gearInRelative.jerk := -1.0;
   cmMasterVirtualAxisX.commandConfiguration.gearInRelative.ratioChangeOnTheFly := FALSE;
   cmMasterVirtualAxisX.commandConfiguration.gearInAbsolute.ratioNumerator := 1;
   cmMasterVirtualAxisX.commandConfiguration.gearInAbsolute.ratioDenominator := 1;
   cmMasterVirtualAxisX.commandConfiguration.gearInAbsolute.masterSyncPosition := 0.0;
   cmMasterVirtualAxisX.commandConfiguration.gearInAbsolute.slaveSyncPosition := 0.0;
   cmMasterVirtualAxisX.commandConfiguration.gearInAbsolute.syncProfileReference := 1;
   cmMasterVirtualAxisX.commandConfiguration.gearInAbsolute.masterStartDistance := 0.0;
   cmMasterVirtualAxisX.commandConfiguration.gearInAbsolute.velocity := -1.0;
   cmMasterVirtualAxisX.commandConfiguration.gearInAbsolute.acceleration := -1.0;
   cmMasterVirtualAxisX.commandConfiguration.gearInAbsolute.deceleration := -1.0;
   cmMasterVirtualAxisX.commandConfiguration.gearInAbsolute.jerk := -1.0;
   cmMasterVirtualAxisX.commandConfiguration.gearInAbsolute.syncDirection := 1;
   cmMasterVirtualAxisX.commandConfiguration.gearInAbsolute.ratioChangeOnTheFly := FALSE;
   cmMasterVirtualAxisX.commandConfiguration.gearInVelocity.continuousUpdate := FALSE;
   cmMasterVirtualAxisX.commandConfiguration.gearInVelocity.ratioNumerator := 1;
   cmMasterVirtualAxisX.commandConfiguration.gearInVelocity.ratioDenominator := 1;
   cmMasterVirtualAxisX.commandConfiguration.gearInVelocity.acceleration := -1.0;
   cmMasterVirtualAxisX.commandConfiguration.gearInVelocity.deceleration := -1.0;
   cmMasterVirtualAxisX.commandConfiguration.gearInVelocity.jerk := -1.0;
   cmMasterVirtualAxisX.commandConfiguration.gearInVelocity.positionControlled := FALSE;
   cmMasterVirtualAxisX.commandConfiguration.camIn.masterOffset := 0.0;
   cmMasterVirtualAxisX.commandConfiguration.camIn.slaveOffset := 0.0;
   cmMasterVirtualAxisX.commandConfiguration.camIn.masterScaling := 1.0;
   cmMasterVirtualAxisX.commandConfiguration.camIn.slaveScaling := 1.0;
   cmMasterVirtualAxisX.commandConfiguration.camIn.masterSyncPosition := 0.0;
   cmMasterVirtualAxisX.commandConfiguration.camIn.syncProfileReference := 1;
   cmMasterVirtualAxisX.commandConfiguration.camIn.masterStartDistance := 0.0;
   cmMasterVirtualAxisX.commandConfiguration.camIn.velocity := -1.0;
   cmMasterVirtualAxisX.commandConfiguration.camIn.acceleration := -1.0;
   cmMasterVirtualAxisX.commandConfiguration.camIn.deceleration := -1.0;
   cmMasterVirtualAxisX.commandConfiguration.camIn.jerk := -1.0;
   cmMasterVirtualAxisX.commandConfiguration.camIn.applicationMode := 0;
   cmMasterVirtualAxisX.commandConfiguration.camIn.syncDirection := 1;
   cmMasterVirtualAxisX.commandConfiguration.gearOutCamOut.slavePosition := 0.0;
   cmMasterVirtualAxisX.commandConfiguration.gearOutCamOut.syncProfileReference := 1;
   cmMasterVirtualAxisX.commandConfiguration.gearOutCamOut.masterStopDistance := 0.0;
   cmMasterVirtualAxisX.commandConfiguration.gearOutCamOut.deceleration := -1.0;
   cmMasterVirtualAxisX.commandConfiguration.gearOutCamOut.jerk := -1.0;
   cmMasterVirtualAxisX.commandConfiguration.gearOutCamOut.syncOutDirection := 3;
   cmMasterVirtualAxisX.commandConfiguration.gearOutCamOut.gearOutCamOutMode := -1;
   cmMasterVirtualAxisX.commandConfiguration.phasing.phaseShift := 0.0;
   cmMasterVirtualAxisX.commandConfiguration.phasing.velocity := -1.0;
   cmMasterVirtualAxisX.commandConfiguration.phasing.acceleration := -1.0;
   cmMasterVirtualAxisX.commandConfiguration.phasing.deceleration := -1.0;
   cmMasterVirtualAxisX.commandConfiguration.phasing.jerk := -1.0;
   cmMasterVirtualAxisX.commandConfiguration.phasing.profileReference := 0;
   cmMasterVirtualAxisX.commandConfiguration.phasing.phasingDistance := 0.0;
   cmMasterVirtualAxisX.commandConfiguration.phasing.startPosition := 0.0;
   cmMasterVirtualAxisX.commandConfiguration.phasing.direction := 3;
   cmMasterVirtualAxisX.commandConfiguration.phasing.phaseAbsolute := TRUE;
   cmMasterVirtualAxisX.commandConfiguration.phasing.phaseShiftChangeOnTheFly := FALSE;
   cmMasterVirtualAxisX.commandConfiguration.offset.offset := 0.0;
   cmMasterVirtualAxisX.commandConfiguration.offset.profileReference := 1;
   cmMasterVirtualAxisX.commandConfiguration.offset.offsetDistance := 0.0;
   cmMasterVirtualAxisX.commandConfiguration.offset.startPosition := 0.0;
   cmMasterVirtualAxisX.commandConfiguration.offset.direction := 3;
   cmMasterVirtualAxisX.commandConfiguration.offset.offsetAbsolute := TRUE;
   cmMasterVirtualAxisX.commandConfiguration.offset.offsetChangeOnTheFly := FALSE;
   cmMasterVirtualAxisX.commands.enableMasterControl := TRUE;
   cmMasterVirtualAxisX.commands.enableAxis := FALSE;
   cmMasterVirtualAxisX.commands.resetAxis := FALSE;
   cmMasterVirtualAxisX.commands.openBrake := FALSE;
   cmMasterVirtualAxisX.commands.jogForward := FALSE;
   cmMasterVirtualAxisX.commands.jogBackward := FALSE;
   cmMasterVirtualAxisX.commands.moveVelocity := FALSE;
   cmMasterVirtualAxisX.commands.stop := FALSE;
   cmMasterVirtualAxisX.commands.fastStop := FALSE;
   cmMasterVirtualAxisX.commands.torqueLimiting := FALSE;
   cmMasterVirtualAxisX.commands.homing := FALSE;
   cmMasterVirtualAxisX.commands.posRelative := FALSE;
   cmMasterVirtualAxisX.commands.posAbsolute := FALSE;
   cmMasterVirtualAxisX.commands.posSuperimposed := FALSE;
   cmMasterVirtualAxisX.commands.haltSuperimposed := FALSE;
   cmMasterVirtualAxisX.commands.selectSetPosition := -1;
   cmMasterVirtualAxisX.commands.uploadParameters := FALSE;
   cmMasterVirtualAxisX.commands.refreshConfiguration := FALSE;
   cmMasterVirtualAxisX.commands.editConfiguration := FALSE;
   cmMasterVirtualAxisX.commands.saveConfiguration := FALSE;
   cmMasterVirtualAxisX.commands.uploadCurrentTorque := FALSE;
   cmMasterVirtualAxisX.commands.reset := FALSE;
   cmMasterVirtualAxisX.monitoring.enable := TRUE;
   cmMasterVirtualAxisX.monitoring.referenceDesignator := WSTRING#'FinalRollerFrontAxisX';
   cmMasterVirtualAxisX.monitoring.enabled := TRUE;
   cmMasterVirtualAxisX.monitoring.enableManualCmds := FALSE;
   cmMasterVirtualAxisX.monitoring.reset := FALSE;
   cmMasterVirtualAxisX.monitoring.resetAxis := FALSE;
   cmMasterVirtualAxisX.monitoring.enableAxis := TRUE;
   cmMasterVirtualAxisX.monitoring.openBrake := FALSE;
   cmMasterVirtualAxisX.monitoring.jogBackward := FALSE;
   cmMasterVirtualAxisX.monitoring.jogForward := FALSE;
   cmMasterVirtualAxisX.monitoring.moveVelocity := FALSE;
   cmMasterVirtualAxisX.monitoring.stop := FALSE;
   cmMasterVirtualAxisX.monitoring.fastStop := FALSE;
   cmMasterVirtualAxisX.monitoring.torqueLimiting := FALSE;
   cmMasterVirtualAxisX.monitoring.homing := FALSE;
   cmMasterVirtualAxisX.monitoring.posRelative := FALSE;
   cmMasterVirtualAxisX.monitoring.posAbsolute := FALSE;
   cmMasterVirtualAxisX.monitoring.posSuperimposed := FALSE;
   cmMasterVirtualAxisX.monitoring.haltSuperimposed := FALSE;
   cmMasterVirtualAxisX.monitoring.brakeOpened := FALSE;
   cmMasterVirtualAxisX.monitoring.axisEnabled := TRUE;
   cmMasterVirtualAxisX.monitoring.resetActive := FALSE;
   cmMasterVirtualAxisX.monitoring.inVelocity := FALSE;
   cmMasterVirtualAxisX.monitoring.inLimitation := FALSE;
   cmMasterVirtualAxisX.monitoring.inClamping := FALSE;
   cmMasterVirtualAxisX.monitoring.startSync := FALSE;
   cmMasterVirtualAxisX.monitoring.inSync := FALSE;
   cmMasterVirtualAxisX.monitoring.inSimulation := FALSE;
   cmMasterVirtualAxisX.monitoring.jogSelected := FALSE;
   cmMasterVirtualAxisX.monitoring.moveVelocitySelected := FALSE;
   cmMasterVirtualAxisX.monitoring.stopSelected := FALSE;
   cmMasterVirtualAxisX.monitoring.fastStopSelected := FALSE;
   cmMasterVirtualAxisX.monitoring.torqueLimitingSelected := FALSE;
   cmMasterVirtualAxisX.monitoring.homingSelected := FALSE;
   cmMasterVirtualAxisX.monitoring.posRelativeSelected := FALSE;
   cmMasterVirtualAxisX.monitoring.posAbsoluteSelected := FALSE;
   cmMasterVirtualAxisX.monitoring.posSuperimposedSelected := FALSE;
   cmMasterVirtualAxisX.monitoring.haltSuperimposedSelected := FALSE;
   cmMasterVirtualAxisX.monitoring.commandBusy := FALSE;
   cmMasterVirtualAxisX.monitoring.commandDone := FALSE;
   cmMasterVirtualAxisX.monitoring.commandAborted := FALSE;
   cmMasterVirtualAxisX.monitoring.homingCommandBusy := FALSE;
   cmMasterVirtualAxisX.monitoring.homingCommandDone := FALSE;
   cmMasterVirtualAxisX.monitoring.homingCommandAborted := FALSE;
   cmMasterVirtualAxisX.monitoring.superimposedBusy := FALSE;
   cmMasterVirtualAxisX.monitoring.superimposedDone := FALSE;
   cmMasterVirtualAxisX.monitoring.superimposedAborted := FALSE;
   cmMasterVirtualAxisX.monitoring.selectSetPosition := -1;
   cmMasterVirtualAxisX.monitoring.selectionController := FALSE;
   cmMasterVirtualAxisX.monitoring.interlockGeneral := TRUE;
   cmMasterVirtualAxisX.monitoring.interlockJogForward := TRUE;
   cmMasterVirtualAxisX.monitoring.interlockJogBackward := TRUE;
   cmMasterVirtualAxisX.monitoring.interlockWarningGeneral := FALSE;
   cmMasterVirtualAxisX.monitoring.interlockWarningJogForward := FALSE;
   cmMasterVirtualAxisX.monitoring.interlockWarningJogBackward := FALSE;
   cmMasterVirtualAxisX.monitoring.valid := TRUE;
   cmMasterVirtualAxisX.monitoring.busy := TRUE;
   cmMasterVirtualAxisX.monitoring.error := TRUE;
   cmMasterVirtualAxisX.monitoring.status := 16#8210;
   cmMasterVirtualAxisX.monitoring.subfunctionStatus := 16#0000;
   cmMasterVirtualAxisX.monitoring.actualPosition := 300919.645;
   cmMasterVirtualAxisX.monitoring.actualSpeed := 325.52;
   cmMasterVirtualAxisX.monitoring.speedUnit := 0;
   cmMasterVirtualAxisX.monitoring.positionUnit := 0;
   cmMasterVirtualAxisX.monitoring.axisStatus1 := 16#0200_1121;
   cmMasterVirtualAxisX.monitoring.axisStatus2 := 16#0000_0000;
   cmMasterVirtualAxisX.monitoring.axisType := -1;
   cmMasterVirtualAxisX.monitoring.maxVelocity := 500.0;
   cmMasterVirtualAxisX.monitoring.actualCurrent := 0.0;
   cmMasterVirtualAxisX.monitoring.actualTorque := 0.0;
   cmMasterVirtualAxisX.monitoring.velocityOverrideEnabled := FALSE;
   cmMasterVirtualAxisX.monitoring.sinaParaError := FALSE;
   cmMasterVirtualAxisX.monitoring.sinaParaStatus := 16#0000_0000;
   cmMasterVirtualAxisX.configuration.referenceDesignator := WSTRING#'FinalRollerFrontAxisX';
   cmMasterVirtualAxisX.configuration.disableAlarms := FALSE;
   cmMasterVirtualAxisX.configuration.masterControlPopUp := TRUE;
   cmMasterVirtualAxisX.configuration.setPositions[0..15].position := 0.0;
   cmMasterVirtualAxisX.configuration.setPositions[0..15].velocity := -1.0;
   cmMasterVirtualAxisX.configuration.setPositions[0..15].acceleration := -1.0;
   cmMasterVirtualAxisX.configuration.setPositions[0..15].deceleration := -1.0;
   cmMasterVirtualAxisX.configuration.setPositions[0..15]."name" := '';
   cmFinalRollerFrontAxisX.commandConfiguration.generalSettings.stopOnError := TRUE;
   cmFinalRollerFrontAxisX.commandConfiguration.generalSettings.resetWithRestart := FALSE;
   cmFinalRollerFrontAxisX.commandConfiguration.generalSettings.abortWaitingSyncCmd := TRUE;
   cmFinalRollerFrontAxisX.commandConfiguration.power.startMode := 1;
   cmFinalRollerFrontAxisX.commandConfiguration.power.stopMode := 0;
   cmFinalRollerFrontAxisX.commandConfiguration.power.syncMotionSimulation := FALSE;
   cmFinalRollerFrontAxisX.commandConfiguration.power.syncMotionSimulationExtendedMode := -1;
   cmFinalRollerFrontAxisX.commandConfiguration.jog.velocity := 0.0;
   cmFinalRollerFrontAxisX.commandConfiguration.jog.acceleration := -1.0;
   cmFinalRollerFrontAxisX.commandConfiguration.jog.deceleration := -1.0;
   cmFinalRollerFrontAxisX.commandConfiguration.jog.jerk := -1.0;
   cmFinalRollerFrontAxisX.commandConfiguration.jog.positionControlled := TRUE;
   cmFinalRollerFrontAxisX.commandConfiguration.jog.increment := 0.0;
   cmFinalRollerFrontAxisX.commandConfiguration.jog.mode := 0;
   cmFinalRollerFrontAxisX.commandConfiguration.moveVelocity.velocity := 0.0;
   cmFinalRollerFrontAxisX.commandConfiguration.moveVelocity.acceleration := -1.0;
   cmFinalRollerFrontAxisX.commandConfiguration.moveVelocity.deceleration := -1.0;
   cmFinalRollerFrontAxisX.commandConfiguration.moveVelocity.jerk := -1.0;
   cmFinalRollerFrontAxisX.commandConfiguration.moveVelocity.direction := 0;
   cmFinalRollerFrontAxisX.commandConfiguration.moveVelocity.positionControlled := TRUE;
   cmFinalRollerFrontAxisX.commandConfiguration.moveVelocity.velocityChangeOnTheFly := FALSE;
   cmFinalRollerFrontAxisX.commandConfiguration.stop.deceleration := -1.0;
   cmFinalRollerFrontAxisX.commandConfiguration.stop.jerk := -1.0;
   cmFinalRollerFrontAxisX.commandConfiguration.stop.abortAcceleration := FALSE;
   cmFinalRollerFrontAxisX.commandConfiguration.fastStop.deceleration := -1.0;
   cmFinalRollerFrontAxisX.commandConfiguration.fastStop.jerk := -1.0;
   cmFinalRollerFrontAxisX.commandConfiguration.fastStop.abortAcceleration := FALSE;
   cmFinalRollerFrontAxisX.commandConfiguration.fastStop.replaceStopPossible := FALSE;
   cmFinalRollerFrontAxisX.commandConfiguration.torqueLimiting.limit := -1.0;
   cmFinalRollerFrontAxisX.commandConfiguration.torqueLimiting.mode := 0;
   cmFinalRollerFrontAxisX.commandConfiguration.homing.position := 0.0;
   cmFinalRollerFrontAxisX.commandConfiguration.homing.mode := 0;
   cmFinalRollerFrontAxisX.commandConfiguration.homing.sensor := 0;
   cmFinalRollerFrontAxisX.commandConfiguration.homing.extendedMode := -1;
   cmFinalRollerFrontAxisX.commandConfiguration.homing.extendedModeTorqueLimit := 0.0;
   cmFinalRollerFrontAxisX.commandConfiguration.homing.extendedModeTargetPosition := 0.0;
   cmFinalRollerFrontAxisX.commandConfiguration.posRelative.distance := 0.0;
   cmFinalRollerFrontAxisX.commandConfiguration.posRelative.velocity := -1.0;
   cmFinalRollerFrontAxisX.commandConfiguration.posRelative.acceleration := -1.0;
   cmFinalRollerFrontAxisX.commandConfiguration.posRelative.deceleration := -1.0;
   cmFinalRollerFrontAxisX.commandConfiguration.posRelative.jerk := -1.0;
   cmFinalRollerFrontAxisX.commandConfiguration.posRelative.direction := 0;
   cmFinalRollerFrontAxisX.commandConfiguration.posAbsolute.position := 0.0;
   cmFinalRollerFrontAxisX.commandConfiguration.posAbsolute.velocity := -1.0;
   cmFinalRollerFrontAxisX.commandConfiguration.posAbsolute.acceleration := -1.0;
   cmFinalRollerFrontAxisX.commandConfiguration.posAbsolute.deceleration := -1.0;
   cmFinalRollerFrontAxisX.commandConfiguration.posAbsolute.jerk := -1.0;
   cmFinalRollerFrontAxisX.commandConfiguration.posAbsolute.direction := 1;
   cmFinalRollerFrontAxisX.commandConfiguration.posAbsolute.positionChangeOnTheFly := FALSE;
   cmFinalRollerFrontAxisX.commandConfiguration.posAbsolute.velocityChangeOnTheFly := FALSE;
   cmFinalRollerFrontAxisX.commandConfiguration.posSuperimposed.distance := 0.0;
   cmFinalRollerFrontAxisX.commandConfiguration.posSuperimposed.velocityDiff := -1.0;
   cmFinalRollerFrontAxisX.commandConfiguration.posSuperimposed.acceleration := -1.0;
   cmFinalRollerFrontAxisX.commandConfiguration.posSuperimposed.deceleration := -1.0;
   cmFinalRollerFrontAxisX.commandConfiguration.posSuperimposed.jerk := -1.0;
   cmFinalRollerFrontAxisX.commandConfiguration.posSuperimposed.direction := 0;
   cmFinalRollerFrontAxisX.commandConfiguration.haltSuperimposed.deceleration := -1.0;
   cmFinalRollerFrontAxisX.commandConfiguration.haltSuperimposed.jerk := -1.0;
   cmFinalRollerFrontAxisX.commandConfiguration.haltSuperimposed.abortAcceleration := FALSE;
   cmFinalRollerFrontAxisX.commandConfiguration.gearInRelative.ratioNumerator := 1;
   cmFinalRollerFrontAxisX.commandConfiguration.gearInRelative.ratioDenominator := 1;
   cmFinalRollerFrontAxisX.commandConfiguration.gearInRelative.acceleration := -1.0;
   cmFinalRollerFrontAxisX.commandConfiguration.gearInRelative.deceleration := -1.0;
   cmFinalRollerFrontAxisX.commandConfiguration.gearInRelative.jerk := -1.0;
   cmFinalRollerFrontAxisX.commandConfiguration.gearInRelative.ratioChangeOnTheFly := FALSE;
   cmFinalRollerFrontAxisX.commandConfiguration.gearInAbsolute.ratioNumerator := 1;
   cmFinalRollerFrontAxisX.commandConfiguration.gearInAbsolute.ratioDenominator := 1;
   cmFinalRollerFrontAxisX.commandConfiguration.gearInAbsolute.masterSyncPosition := 0.0;
   cmFinalRollerFrontAxisX.commandConfiguration.gearInAbsolute.slaveSyncPosition := 0.0;
   cmFinalRollerFrontAxisX.commandConfiguration.gearInAbsolute.syncProfileReference := 1;
   cmFinalRollerFrontAxisX.commandConfiguration.gearInAbsolute.masterStartDistance := 0.0;
   cmFinalRollerFrontAxisX.commandConfiguration.gearInAbsolute.velocity := -1.0;
   cmFinalRollerFrontAxisX.commandConfiguration.gearInAbsolute.acceleration := -1.0;
   cmFinalRollerFrontAxisX.commandConfiguration.gearInAbsolute.deceleration := -1.0;
   cmFinalRollerFrontAxisX.commandConfiguration.gearInAbsolute.jerk := -1.0;
   cmFinalRollerFrontAxisX.commandConfiguration.gearInAbsolute.syncDirection := 1;
   cmFinalRollerFrontAxisX.commandConfiguration.gearInAbsolute.ratioChangeOnTheFly := FALSE;
   cmFinalRollerFrontAxisX.commandConfiguration.gearInVelocity.continuousUpdate := FALSE;
   cmFinalRollerFrontAxisX.commandConfiguration.gearInVelocity.ratioNumerator := 1;
   cmFinalRollerFrontAxisX.commandConfiguration.gearInVelocity.ratioDenominator := 1;
   cmFinalRollerFrontAxisX.commandConfiguration.gearInVelocity.acceleration := -1.0;
   cmFinalRollerFrontAxisX.commandConfiguration.gearInVelocity.deceleration := -1.0;
   cmFinalRollerFrontAxisX.commandConfiguration.gearInVelocity.jerk := -1.0;
   cmFinalRollerFrontAxisX.commandConfiguration.gearInVelocity.positionControlled := FALSE;
   cmFinalRollerFrontAxisX.commandConfiguration.camIn.masterOffset := 0.0;
   cmFinalRollerFrontAxisX.commandConfiguration.camIn.slaveOffset := 0.0;
   cmFinalRollerFrontAxisX.commandConfiguration.camIn.masterScaling := 1.0;
   cmFinalRollerFrontAxisX.commandConfiguration.camIn.slaveScaling := 1.0;
   cmFinalRollerFrontAxisX.commandConfiguration.camIn.masterSyncPosition := 0.0;
   cmFinalRollerFrontAxisX.commandConfiguration.camIn.syncProfileReference := 1;
   cmFinalRollerFrontAxisX.commandConfiguration.camIn.masterStartDistance := 0.0;
   cmFinalRollerFrontAxisX.commandConfiguration.camIn.velocity := -1.0;
   cmFinalRollerFrontAxisX.commandConfiguration.camIn.acceleration := -1.0;
   cmFinalRollerFrontAxisX.commandConfiguration.camIn.deceleration := -1.0;
   cmFinalRollerFrontAxisX.commandConfiguration.camIn.jerk := -1.0;
   cmFinalRollerFrontAxisX.commandConfiguration.camIn.applicationMode := 0;
   cmFinalRollerFrontAxisX.commandConfiguration.camIn.syncDirection := 1;
   cmFinalRollerFrontAxisX.commandConfiguration.gearOutCamOut.slavePosition := 0.0;
   cmFinalRollerFrontAxisX.commandConfiguration.gearOutCamOut.syncProfileReference := 1;
   cmFinalRollerFrontAxisX.commandConfiguration.gearOutCamOut.masterStopDistance := 0.0;
   cmFinalRollerFrontAxisX.commandConfiguration.gearOutCamOut.deceleration := -1.0;
   cmFinalRollerFrontAxisX.commandConfiguration.gearOutCamOut.jerk := -1.0;
   cmFinalRollerFrontAxisX.commandConfiguration.gearOutCamOut.syncOutDirection := 3;
   cmFinalRollerFrontAxisX.commandConfiguration.gearOutCamOut.gearOutCamOutMode := -1;
   cmFinalRollerFrontAxisX.commandConfiguration.phasing.phaseShift := 0.0;
   cmFinalRollerFrontAxisX.commandConfiguration.phasing.velocity := -1.0;
   cmFinalRollerFrontAxisX.commandConfiguration.phasing.acceleration := -1.0;
   cmFinalRollerFrontAxisX.commandConfiguration.phasing.deceleration := -1.0;
   cmFinalRollerFrontAxisX.commandConfiguration.phasing.jerk := -1.0;
   cmFinalRollerFrontAxisX.commandConfiguration.phasing.profileReference := 0;
   cmFinalRollerFrontAxisX.commandConfiguration.phasing.phasingDistance := 0.0;
   cmFinalRollerFrontAxisX.commandConfiguration.phasing.startPosition := 0.0;
   cmFinalRollerFrontAxisX.commandConfiguration.phasing.direction := 3;
   cmFinalRollerFrontAxisX.commandConfiguration.phasing.phaseAbsolute := TRUE;
   cmFinalRollerFrontAxisX.commandConfiguration.phasing.phaseShiftChangeOnTheFly := FALSE;
   cmFinalRollerFrontAxisX.commandConfiguration.offset.offset := 0.0;
   cmFinalRollerFrontAxisX.commandConfiguration.offset.profileReference := 1;
   cmFinalRollerFrontAxisX.commandConfiguration.offset.offsetDistance := 0.0;
   cmFinalRollerFrontAxisX.commandConfiguration.offset.startPosition := 0.0;
   cmFinalRollerFrontAxisX.commandConfiguration.offset.direction := 3;
   cmFinalRollerFrontAxisX.commandConfiguration.offset.offsetAbsolute := TRUE;
   cmFinalRollerFrontAxisX.commandConfiguration.offset.offsetChangeOnTheFly := FALSE;
   cmFinalRollerFrontAxisX.commands.enableMasterControl := TRUE;
   cmFinalRollerFrontAxisX.commands.enableAxis := FALSE;
   cmFinalRollerFrontAxisX.commands.resetAxis := FALSE;
   cmFinalRollerFrontAxisX.commands.openBrake := FALSE;
   cmFinalRollerFrontAxisX.commands.jogForward := FALSE;
   cmFinalRollerFrontAxisX.commands.jogBackward := FALSE;
   cmFinalRollerFrontAxisX.commands.moveVelocity := FALSE;
   cmFinalRollerFrontAxisX.commands.stop := FALSE;
   cmFinalRollerFrontAxisX.commands.fastStop := FALSE;
   cmFinalRollerFrontAxisX.commands.torqueLimiting := FALSE;
   cmFinalRollerFrontAxisX.commands.homing := FALSE;
   cmFinalRollerFrontAxisX.commands.posRelative := FALSE;
   cmFinalRollerFrontAxisX.commands.posAbsolute := FALSE;
   cmFinalRollerFrontAxisX.commands.posSuperimposed := FALSE;
   cmFinalRollerFrontAxisX.commands.haltSuperimposed := FALSE;
   cmFinalRollerFrontAxisX.commands.selectSetPosition := 0;
   cmFinalRollerFrontAxisX.commands.uploadParameters := FALSE;
   cmFinalRollerFrontAxisX.commands.refreshConfiguration := FALSE;
   cmFinalRollerFrontAxisX.commands.editConfiguration := FALSE;
   cmFinalRollerFrontAxisX.commands.saveConfiguration := FALSE;
   cmFinalRollerFrontAxisX.commands.uploadCurrentTorque := FALSE;
   cmFinalRollerFrontAxisX.commands.reset := FALSE;
   cmFinalRollerFrontAxisX.monitoring.enable := TRUE;
   cmFinalRollerFrontAxisX.monitoring.referenceDesignator := WSTRING#'FinalRollerFrontAxisX';
   cmFinalRollerFrontAxisX.monitoring.enabled := TRUE;
   cmFinalRollerFrontAxisX.monitoring.enableManualCmds := FALSE;
   cmFinalRollerFrontAxisX.monitoring.reset := FALSE;
   cmFinalRollerFrontAxisX.monitoring.resetAxis := FALSE;
   cmFinalRollerFrontAxisX.monitoring.enableAxis := TRUE;
   cmFinalRollerFrontAxisX.monitoring.openBrake := FALSE;
   cmFinalRollerFrontAxisX.monitoring.jogBackward := FALSE;
   cmFinalRollerFrontAxisX.monitoring.jogForward := FALSE;
   cmFinalRollerFrontAxisX.monitoring.moveVelocity := FALSE;
   cmFinalRollerFrontAxisX.monitoring.stop := FALSE;
   cmFinalRollerFrontAxisX.monitoring.fastStop := FALSE;
   cmFinalRollerFrontAxisX.monitoring.torqueLimiting := FALSE;
   cmFinalRollerFrontAxisX.monitoring.homing := FALSE;
   cmFinalRollerFrontAxisX.monitoring.posRelative := FALSE;
   cmFinalRollerFrontAxisX.monitoring.posAbsolute := FALSE;
   cmFinalRollerFrontAxisX.monitoring.posSuperimposed := FALSE;
   cmFinalRollerFrontAxisX.monitoring.haltSuperimposed := FALSE;
   cmFinalRollerFrontAxisX.monitoring.brakeOpened := FALSE;
   cmFinalRollerFrontAxisX.monitoring.axisEnabled := TRUE;
   cmFinalRollerFrontAxisX.monitoring.resetActive := FALSE;
   cmFinalRollerFrontAxisX.monitoring.inVelocity := FALSE;
   cmFinalRollerFrontAxisX.monitoring.inLimitation := FALSE;
   cmFinalRollerFrontAxisX.monitoring.inClamping := FALSE;
   cmFinalRollerFrontAxisX.monitoring.startSync := FALSE;
   cmFinalRollerFrontAxisX.monitoring.inSync := FALSE;
   cmFinalRollerFrontAxisX.monitoring.inSimulation := FALSE;
   cmFinalRollerFrontAxisX.monitoring.jogSelected := FALSE;
   cmFinalRollerFrontAxisX.monitoring.moveVelocitySelected := FALSE;
   cmFinalRollerFrontAxisX.monitoring.stopSelected := FALSE;
   cmFinalRollerFrontAxisX.monitoring.fastStopSelected := FALSE;
   cmFinalRollerFrontAxisX.monitoring.torqueLimitingSelected := FALSE;
   cmFinalRollerFrontAxisX.monitoring.homingSelected := FALSE;
   cmFinalRollerFrontAxisX.monitoring.posRelativeSelected := FALSE;
   cmFinalRollerFrontAxisX.monitoring.posAbsoluteSelected := FALSE;
   cmFinalRollerFrontAxisX.monitoring.posSuperimposedSelected := FALSE;
   cmFinalRollerFrontAxisX.monitoring.haltSuperimposedSelected := FALSE;
   cmFinalRollerFrontAxisX.monitoring.commandBusy := FALSE;
   cmFinalRollerFrontAxisX.monitoring.commandDone := FALSE;
   cmFinalRollerFrontAxisX.monitoring.commandAborted := FALSE;
   cmFinalRollerFrontAxisX.monitoring.homingCommandBusy := FALSE;
   cmFinalRollerFrontAxisX.monitoring.homingCommandDone := FALSE;
   cmFinalRollerFrontAxisX.monitoring.homingCommandAborted := FALSE;
   cmFinalRollerFrontAxisX.monitoring.superimposedBusy := FALSE;
   cmFinalRollerFrontAxisX.monitoring.superimposedDone := FALSE;
   cmFinalRollerFrontAxisX.monitoring.superimposedAborted := FALSE;
   cmFinalRollerFrontAxisX.monitoring.selectSetPosition := 0;
   cmFinalRollerFrontAxisX.monitoring.selectionController := FALSE;
   cmFinalRollerFrontAxisX.monitoring.interlockGeneral := TRUE;
   cmFinalRollerFrontAxisX.monitoring.interlockJogForward := TRUE;
   cmFinalRollerFrontAxisX.monitoring.interlockJogBackward := TRUE;
   cmFinalRollerFrontAxisX.monitoring.interlockWarningGeneral := FALSE;
   cmFinalRollerFrontAxisX.monitoring.interlockWarningJogForward := FALSE;
   cmFinalRollerFrontAxisX.monitoring.interlockWarningJogBackward := FALSE;
   cmFinalRollerFrontAxisX.monitoring.valid := TRUE;
   cmFinalRollerFrontAxisX.monitoring.busy := TRUE;
   cmFinalRollerFrontAxisX.monitoring.error := FALSE;
   cmFinalRollerFrontAxisX.monitoring.status := 16#7002;
   cmFinalRollerFrontAxisX.monitoring.subfunctionStatus := 16#0000;
   cmFinalRollerFrontAxisX.monitoring.actualPosition := 273.643;
   cmFinalRollerFrontAxisX.monitoring.actualSpeed := 696.958289998712;
   cmFinalRollerFrontAxisX.monitoring.speedUnit := 1062;
   cmFinalRollerFrontAxisX.monitoring.positionUnit := 1013;
   cmFinalRollerFrontAxisX.monitoring.axisStatus1 := 16#0240_4021;
   cmFinalRollerFrontAxisX.monitoring.axisStatus2 := 16#0000_0000;
   cmFinalRollerFrontAxisX.monitoring.axisType := 1;
   cmFinalRollerFrontAxisX.monitoring.maxVelocity := 2500.0;
   cmFinalRollerFrontAxisX.monitoring.actualCurrent := 0.0;
   cmFinalRollerFrontAxisX.monitoring.actualTorque := 0.0;
   cmFinalRollerFrontAxisX.monitoring.velocityOverrideEnabled := FALSE;
   cmFinalRollerFrontAxisX.monitoring.sinaParaError := FALSE;
   cmFinalRollerFrontAxisX.monitoring.sinaParaStatus := 16#0000_0000;
   cmFinalRollerFrontAxisX.configuration.referenceDesignator := WSTRING#'FinalRollerFrontAxisX';
   cmFinalRollerFrontAxisX.configuration.disableAlarms := FALSE;
   cmFinalRollerFrontAxisX.configuration.masterControlPopUp := TRUE;
   cmFinalRollerFrontAxisX.configuration.setPositions[0].position := 0.0;
   cmFinalRollerFrontAxisX.configuration.setPositions[1].position := 500.0;
   cmFinalRollerFrontAxisX.configuration.setPositions[2..15].position := 0.0;
   cmFinalRollerFrontAxisX.configuration.setPositions[0..1].velocity := 500.0;
   cmFinalRollerFrontAxisX.configuration.setPositions[2..15].velocity := -1.0;
   cmFinalRollerFrontAxisX.configuration.setPositions[0..1].acceleration := 5000.0;
   cmFinalRollerFrontAxisX.configuration.setPositions[2..15].acceleration := -1.0;
   cmFinalRollerFrontAxisX.configuration.setPositions[0..1].deceleration := 5000.0;
   cmFinalRollerFrontAxisX.configuration.setPositions[2..15].deceleration := -1.0;
   cmFinalRollerFrontAxisX.configuration.setPositions[0..15]."name" := '';
   cmFinalRollerRearAxisX.commandConfiguration.generalSettings.stopOnError := TRUE;
   cmFinalRollerRearAxisX.commandConfiguration.generalSettings.resetWithRestart := FALSE;
   cmFinalRollerRearAxisX.commandConfiguration.generalSettings.abortWaitingSyncCmd := TRUE;
   cmFinalRollerRearAxisX.commandConfiguration.power.startMode := 1;
   cmFinalRollerRearAxisX.commandConfiguration.power.stopMode := 0;
   cmFinalRollerRearAxisX.commandConfiguration.power.syncMotionSimulation := FALSE;
   cmFinalRollerRearAxisX.commandConfiguration.power.syncMotionSimulationExtendedMode := -1;
   cmFinalRollerRearAxisX.commandConfiguration.jog.velocity := 0.0;
   cmFinalRollerRearAxisX.commandConfiguration.jog.acceleration := -1.0;
   cmFinalRollerRearAxisX.commandConfiguration.jog.deceleration := -1.0;
   cmFinalRollerRearAxisX.commandConfiguration.jog.jerk := -1.0;
   cmFinalRollerRearAxisX.commandConfiguration.jog.positionControlled := TRUE;
   cmFinalRollerRearAxisX.commandConfiguration.jog.increment := 0.0;
   cmFinalRollerRearAxisX.commandConfiguration.jog.mode := 0;
   cmFinalRollerRearAxisX.commandConfiguration.moveVelocity.velocity := 0.0;
   cmFinalRollerRearAxisX.commandConfiguration.moveVelocity.acceleration := -1.0;
   cmFinalRollerRearAxisX.commandConfiguration.moveVelocity.deceleration := -1.0;
   cmFinalRollerRearAxisX.commandConfiguration.moveVelocity.jerk := -1.0;
   cmFinalRollerRearAxisX.commandConfiguration.moveVelocity.direction := 0;
   cmFinalRollerRearAxisX.commandConfiguration.moveVelocity.positionControlled := TRUE;
   cmFinalRollerRearAxisX.commandConfiguration.moveVelocity.velocityChangeOnTheFly := FALSE;
   cmFinalRollerRearAxisX.commandConfiguration.stop.deceleration := -1.0;
   cmFinalRollerRearAxisX.commandConfiguration.stop.jerk := -1.0;
   cmFinalRollerRearAxisX.commandConfiguration.stop.abortAcceleration := FALSE;
   cmFinalRollerRearAxisX.commandConfiguration.fastStop.deceleration := -1.0;
   cmFinalRollerRearAxisX.commandConfiguration.fastStop.jerk := -1.0;
   cmFinalRollerRearAxisX.commandConfiguration.fastStop.abortAcceleration := FALSE;
   cmFinalRollerRearAxisX.commandConfiguration.fastStop.replaceStopPossible := FALSE;
   cmFinalRollerRearAxisX.commandConfiguration.torqueLimiting.limit := -1.0;
   cmFinalRollerRearAxisX.commandConfiguration.torqueLimiting.mode := 0;
   cmFinalRollerRearAxisX.commandConfiguration.homing.position := 0.0;
   cmFinalRollerRearAxisX.commandConfiguration.homing.mode := 0;   // Homing Mode
   cmFinalRollerRearAxisX.commandConfiguration.homing.sensor := 0;
   cmFinalRollerRearAxisX.commandConfiguration.homing.extendedMode := -1;
   cmFinalRollerRearAxisX.commandConfiguration.homing.extendedModeTorqueLimit := 0.0;
   cmFinalRollerRearAxisX.commandConfiguration.homing.extendedModeTargetPosition := 0.0;
   cmFinalRollerRearAxisX.commandConfiguration.posRelative.distance := 0.0;
   cmFinalRollerRearAxisX.commandConfiguration.posRelative.velocity := -1.0;
   cmFinalRollerRearAxisX.commandConfiguration.posRelative.acceleration := -1.0;
   cmFinalRollerRearAxisX.commandConfiguration.posRelative.deceleration := -1.0;
   cmFinalRollerRearAxisX.commandConfiguration.posRelative.jerk := -1.0;
   cmFinalRollerRearAxisX.commandConfiguration.posRelative.direction := 0;
   cmFinalRollerRearAxisX.commandConfiguration.posAbsolute.position := 0.0;
   cmFinalRollerRearAxisX.commandConfiguration.posAbsolute.velocity := -1.0;
   cmFinalRollerRearAxisX.commandConfiguration.posAbsolute.acceleration := -1.0;
   cmFinalRollerRearAxisX.commandConfiguration.posAbsolute.deceleration := -1.0;
   cmFinalRollerRearAxisX.commandConfiguration.posAbsolute.jerk := -1.0;
   cmFinalRollerRearAxisX.commandConfiguration.posAbsolute.direction := 1;
   cmFinalRollerRearAxisX.commandConfiguration.posAbsolute.positionChangeOnTheFly := FALSE;
   cmFinalRollerRearAxisX.commandConfiguration.posAbsolute.velocityChangeOnTheFly := FALSE;
   cmFinalRollerRearAxisX.commandConfiguration.posSuperimposed.distance := 0.0;
   cmFinalRollerRearAxisX.commandConfiguration.posSuperimposed.velocityDiff := -1.0;
   cmFinalRollerRearAxisX.commandConfiguration.posSuperimposed.acceleration := -1.0;
   cmFinalRollerRearAxisX.commandConfiguration.posSuperimposed.deceleration := -1.0;
   cmFinalRollerRearAxisX.commandConfiguration.posSuperimposed.jerk := -1.0;
   cmFinalRollerRearAxisX.commandConfiguration.posSuperimposed.direction := 0;
   cmFinalRollerRearAxisX.commandConfiguration.haltSuperimposed.deceleration := -1.0;
   cmFinalRollerRearAxisX.commandConfiguration.haltSuperimposed.jerk := -1.0;
   cmFinalRollerRearAxisX.commandConfiguration.haltSuperimposed.abortAcceleration := FALSE;
   cmFinalRollerRearAxisX.commandConfiguration.gearInRelative.ratioNumerator := 1;
   cmFinalRollerRearAxisX.commandConfiguration.gearInRelative.ratioDenominator := 1;
   cmFinalRollerRearAxisX.commandConfiguration.gearInRelative.acceleration := -1.0;
   cmFinalRollerRearAxisX.commandConfiguration.gearInRelative.deceleration := -1.0;
   cmFinalRollerRearAxisX.commandConfiguration.gearInRelative.jerk := -1.0;
   cmFinalRollerRearAxisX.commandConfiguration.gearInRelative.ratioChangeOnTheFly := FALSE;
   cmFinalRollerRearAxisX.commandConfiguration.gearInAbsolute.ratioNumerator := 1;
   cmFinalRollerRearAxisX.commandConfiguration.gearInAbsolute.ratioDenominator := 1;
   cmFinalRollerRearAxisX.commandConfiguration.gearInAbsolute.masterSyncPosition := 0.0;
   cmFinalRollerRearAxisX.commandConfiguration.gearInAbsolute.slaveSyncPosition := 0.0;
   cmFinalRollerRearAxisX.commandConfiguration.gearInAbsolute.syncProfileReference := 1;
   cmFinalRollerRearAxisX.commandConfiguration.gearInAbsolute.masterStartDistance := 0.0;
   cmFinalRollerRearAxisX.commandConfiguration.gearInAbsolute.velocity := -1.0;
   cmFinalRollerRearAxisX.commandConfiguration.gearInAbsolute.acceleration := -1.0;
   cmFinalRollerRearAxisX.commandConfiguration.gearInAbsolute.deceleration := -1.0;
   cmFinalRollerRearAxisX.commandConfiguration.gearInAbsolute.jerk := -1.0;
   cmFinalRollerRearAxisX.commandConfiguration.gearInAbsolute.syncDirection := 1;
   cmFinalRollerRearAxisX.commandConfiguration.gearInAbsolute.ratioChangeOnTheFly := FALSE;
   cmFinalRollerRearAxisX.commandConfiguration.gearInVelocity.continuousUpdate := FALSE;
   cmFinalRollerRearAxisX.commandConfiguration.gearInVelocity.ratioNumerator := 1;
   cmFinalRollerRearAxisX.commandConfiguration.gearInVelocity.ratioDenominator := 1;
   cmFinalRollerRearAxisX.commandConfiguration.gearInVelocity.acceleration := -1.0;
   cmFinalRollerRearAxisX.commandConfiguration.gearInVelocity.deceleration := -1.0;
   cmFinalRollerRearAxisX.commandConfiguration.gearInVelocity.jerk := -1.0;
   cmFinalRollerRearAxisX.commandConfiguration.gearInVelocity.positionControlled := FALSE;
   cmFinalRollerRearAxisX.commandConfiguration.camIn.masterOffset := 0.0;
   cmFinalRollerRearAxisX.commandConfiguration.camIn.slaveOffset := 0.0;
   cmFinalRollerRearAxisX.commandConfiguration.camIn.masterScaling := 1.0;
   cmFinalRollerRearAxisX.commandConfiguration.camIn.slaveScaling := 1.0;
   cmFinalRollerRearAxisX.commandConfiguration.camIn.masterSyncPosition := 0.0;
   cmFinalRollerRearAxisX.commandConfiguration.camIn.syncProfileReference := 1;
   cmFinalRollerRearAxisX.commandConfiguration.camIn.masterStartDistance := 0.0;
   cmFinalRollerRearAxisX.commandConfiguration.camIn.velocity := -1.0;
   cmFinalRollerRearAxisX.commandConfiguration.camIn.acceleration := -1.0;
   cmFinalRollerRearAxisX.commandConfiguration.camIn.deceleration := -1.0;
   cmFinalRollerRearAxisX.commandConfiguration.camIn.jerk := -1.0;
   cmFinalRollerRearAxisX.commandConfiguration.camIn.applicationMode := 0;
   cmFinalRollerRearAxisX.commandConfiguration.camIn.syncDirection := 1;
   cmFinalRollerRearAxisX.commandConfiguration.gearOutCamOut.slavePosition := 0.0;
   cmFinalRollerRearAxisX.commandConfiguration.gearOutCamOut.syncProfileReference := 1;
   cmFinalRollerRearAxisX.commandConfiguration.gearOutCamOut.masterStopDistance := 0.0;
   cmFinalRollerRearAxisX.commandConfiguration.gearOutCamOut.deceleration := -1.0;
   cmFinalRollerRearAxisX.commandConfiguration.gearOutCamOut.jerk := -1.0;
   cmFinalRollerRearAxisX.commandConfiguration.gearOutCamOut.syncOutDirection := 3;
   cmFinalRollerRearAxisX.commandConfiguration.gearOutCamOut.gearOutCamOutMode := -1;
   cmFinalRollerRearAxisX.commandConfiguration.phasing.phaseShift := 0.0;
   cmFinalRollerRearAxisX.commandConfiguration.phasing.velocity := -1.0;
   cmFinalRollerRearAxisX.commandConfiguration.phasing.acceleration := -1.0;
   cmFinalRollerRearAxisX.commandConfiguration.phasing.deceleration := -1.0;
   cmFinalRollerRearAxisX.commandConfiguration.phasing.jerk := -1.0;
   cmFinalRollerRearAxisX.commandConfiguration.phasing.profileReference := 0;
   cmFinalRollerRearAxisX.commandConfiguration.phasing.phasingDistance := 0.0;
   cmFinalRollerRearAxisX.commandConfiguration.phasing.startPosition := 0.0;
   cmFinalRollerRearAxisX.commandConfiguration.phasing.direction := 3;
   cmFinalRollerRearAxisX.commandConfiguration.phasing.phaseAbsolute := TRUE;
